# B&R Automation Studio project TD52 (part 31)

#### TrP_red.st
```iecst
(*******************************************************************************
TransP_red	Powerreduction cause of transformer warning

This code is confidential and proprietary to the INNIO Company.
It may not be used in any form, or reproduced in any manner,
without the express written permission of the INNIO Company.
Copyright, INNIO Company, 2019

Customized modifications: -
------------------------

History:
-------
V4.03.00	24.07.2015	Plattner Johannes
V4.04.00	23.09.2016	lettenb.	OUT_AG.rP_Red_TransformerWarning_Norm: /100 removed, bugfix
			08.05.2017				Pred logic corr., bugfix

Instructions for use:
--------------------

Power reduction from Transformer Warning.
Activates with parameter:		AuxiliariesGeneral::AsGlobalPV.bP_Red_TransformerWarning
Power setpoint with parameter:	AuxiliariesGeneral::AsGlobalPV.rP_Red_TransformerWarning_Rate

Outstandings:
------------
*******************************************************************************)
PROGRAM _CYCLIC

	(* Transformer power reduction aktive*)
	(*----------------------------------------------------------------------------*)
	IF Para.bP_Red_TransformerWarning_Sel AND NOT IN_AG.tTransformerWarning.Di THEN

		OUT_AG.rP_Red_TransformerWarning_Norm	:= LIMIT(0.5, Para.rP_Red_TransformerWarning_Rate,1.0);
		OUT_AG.bP_Red_TransformerWarning_Sel	:= TRUE;
	(*----------------------------------------------------------------------------*)

	(* Transformer power reduction inaktive*)
	(*----------------------------------------------------------------------------*)
	ELSE

		OUT_AG.bP_Red_TransformerWarning_Sel	:= FALSE;
		OUT_AG.rP_Red_TransformerWarning_Norm	:= 1.0;

	END_IF;
	(*----------------------------------------------------------------------------*)

END_PROGRAM
```

### Program Logical/AuxiliariesGeneral/Cnt_EO (IEC, version 4.13.0) - engine oil counter

#### Cnt_EOCyclic.st
```iecst
(***********************************************************************************************************************
AGGR: oil consumption counting and saving data (cyclic)

This code is confidential and proprietary to the INNIO Company.
It may not be used in any form, or reproduced in any manner, without the express
written permission of the INNIO Company.
Copyright, INNIO Company, 2024

- detection of oilcounter impulses
- logging oil volume(ml) and active energy(kwh)

Customized modifications: -
------------------------

History:
-------
V2.0	26.06.2007	TinelloM 	erstellt
V2.1	16.08.2007 	TinelloM 	überarbeitet
V2.3	31.03.2008 	TinelloM	überarbeitet für Serie
V3.20	20.07.2010	KoppM		anpassung für BR9 und analogen Füllstandsensor
V3.20.1	08.02.2011	TinelloM	IF ucIndexOil >1...
V3.90.0	06.12.2011	Ganguly		generated from oilcountCyclic.st V3.20.1
V3.90.1	12.03.2012	Denk		review and clean-up
V3.91	03.09.2013	Zengerer 	BUGFIX in nextline copy : OilCounter[i]	:= OilCounter[i+1];
V3.99.0 04.12.2013	lettenb.	slOilCounterMax,rSumOilVolume,rSumActiveEnergy: conversion dint_to_real added
V4.00.0	03.11.2014	lettenb.	init: DatObjCreate_01.MemType:= doSYSROM --> doUSRROM (vis kann bei update nicht in SYSROM schreiben)
		28.04.2015				set rAvgVolumeEnergy:=0 IF no averaging is selected, bugfix
V4.03.0	03.11.2015	lettenb.	calc. rAvgVolumeEnergy corr., bugfix
		11.01.2016				MM2VIS oil counter interfaces moved from Vis_AG -> Cnt_EO(to enable scroll function of settings)bugfix
		15.02.2016  waldhart	datenpunkte für HMI aus der IF-schleife entfernt(P19 test)
V4.05.0	14.12.2017	lettenb.	IN_AG.rP_Act_Norm_Filt -> IN_AG.rP_Act_Norm_Filt_TC2, mapping cleanup
		27.12.2017				bReset_Bh added, to reset oil counter memory after engine change(iCnt_OpHours -> 0)
V4.06.0 005 11.09.2018 Zengerer	beta: OUT_AG.tAG2PB.bPermSetupOk... new: transmit perm status info in InitUp
V4.07				Zengerer	Do not allow old data file lengt in init, to force rebuild with latest file format !
V4.09.0	09.10.2019	Schmid		BU1: reduced number of perm file write cycles (max every 10min)
V4.10.0	03.12.2020	Perktold,	added oil and coolant management
		25.01.2021	Schmid		bugfix oil refill blockade after iCnt_OpHours reset (engine exchange)
		11.03.2021	lettenb.	9004->9048, Msg# already used, bugfix
V4.11.0	19.01.2022	Schmid		option for oil sampling interval from oil quality sensor
V4.12.0	29.03.2023	Tinello		bugfix #1092 oil counter reset
V4.13.0	13.02.2024	Tinello		oil refill monitoring

Instructions for use:
--------------------
The parameter are stored in a data module which is stored on flash memory.
At start up the parameter will be readed from the flash memory and copied to

Outstandings:
------------
-
***********************************************************************************************************************)

PROGRAM _CYCLIC

(* getting time of the controller *)
	DTGetTime_RPS.enable := TRUE;							(* getting *)
	DTGetTime_RPS();
	DT_TO_DTStructure(DTGetTime_RPS.DT1, ADR(tRealTime));	(* change format *)
	DTGetTime_RPS.status;

	(* oil counter is active *)
	IF Para.b_OilActive THEN

		(* oilcounter impulse detection *)
		xR_TRIG_OilCounterImpulse(CLK := IN_AG.tCnt_OilPulse.Di);
		IF xR_TRIG_OilCounterImpulse.Q THEN  slOilCounterImpulse := slOilCounterImpulse + 1;	END_IF

		(* reset *)
		IF ucResetRegister1 = 0	THEN slOilCounterImpulse := 0;	END_IF

		(* oilcounter impulse detection for X20DC2395 --> Reset not possible *)
		IF REAL_TO_UINT(IN_AG.tCnt_Oil_DC2395.Ai) >= usOilCounterStart	THEN
			slOilCounterCircle	:= (REAL_TO_DINT(IN_AG.tCnt_Oil_DC2395.Ai) - usOilCounterStart) / 2;
		ELSE
			slOilCounterCircle	:= (REAL_TO_DINT(IN_AG.tCnt_Oil_DC2395.Ai) - usOilCounterStart + 65535) / 2;
		END_IF

		(* generate second based clock pulse *)
		xTON_SecondTick(IN := NOT xTON_SecondTick.Q, PT := T#980ms);		(* 980ms + 2 times cycle time = 1 sec.*)

		IF xTON_SecondTick.Q THEN

			(* reset *)
			bErrMsOilCounter	:= FALSE;
			b_OilRefillBlocked	:= FALSE;

			FOR i:=0 TO 19 BY 1 DO
				IF IN_AG.iCnt_OpHours > 0 AND IN_AG.iCnt_OpHours + 10000 < OilCounter[i].Bh THEN bReset_Bh := TRUE; (* reset OpHours(engine change)*)
				END_IF;
			END_FOR;

			(* Delete circular puffer array of oil measurements *)
			IF bReset_Bh THEN
				FOR i:=0 TO 19 BY 1 DO
					OilCounter[i].oil_volume		:= 0;
					OilCounter[i].delta_kwh 		:= 0;
					OilCounter[i].day 				:= 0;
					OilCounter[i].month 			:= 0;
					OilCounter[i].year 				:= 0;
					OilCounter[i].hour 				:= 0;
					OilCounter[i].minute 			:= 0;
					OilCounter[i].averaging			:= 0;
					OilCounter[i].Bh				:= 0;
					OilCounter[i].rOC_Consum		:= 0;
					OilCounter[i].rOC_DeltaOpHour	:= 0;
					OilCounter[i].rP_OC_Avg			:= 0;
				END_FOR

				ucIndexOil 	:= 0;										(* reset circular puffer index	*)
				bReset_Bh	:= FALSE;
			END_IF

			(* Identification of active oil counter input *)
			slOilCounterMax	:= MAX(slOilCounterCircle, slOilCounterImpulse);
			slOilCounterMax	:= REAL_TO_DINT(MAX(DINT_TO_REAL(slOilCounterMax), IN_AG.tCnt_Oil_NC150.Ai));

			slOilCounter	:= slOilCounterMax * 					(* maximum number of oil counter impulses 		*)
						   	   Para.iNum_OilPulse;					(* 1 impulse e.g.=2ml, -> 500 impulses/liter	*)

			(* Oil refill monitoring *)
			rVol_OilRefill_Max		:= (Para.rVol_OilRefill_Pct_EO_Level * 1000)	  *		(* oil refill volume [ml] per % oil level *)
									   (Para.r_OV_LimClose - Para.r_OV_LimOpen) * 100 *		(* % oil level between open- and closing of valve *)
									   (1.0 + Para.rPc_OilRefill_VolTolerance);				(* Tolerance *)

			bAMM_Vol_OilRefill_Hi	:= (slOilCounter > REAL_TO_DINT(rVol_OilRefill_Max)) AND Para.bOilRefill_MonAct AND Para.bEO_Level_Active;		(* W9378 *)

			(* calculation of kilowatt hour *)
			IF (IN_AG.rP_Act_Norm_Filt_TC2 * IN_AG.rP_Nom) > 50	THEN
				kwh	:= kwh + ((IN_AG.rP_Act_Norm_Filt_TC2 * IN_AG.rP_Nom) / 3600 );
			END_IF

			(* When Oilrefillvalve is closed, data will be saved *)
		 	xF_TRIG_OilRefillValve(CLK := OUT_AG.tEOVal_DemOpen.Do);

		 	IF 	xF_TRIG_OilRefillValve.Q	THEN
				(* monitoring measurement signal oil counter *)
				IF slOilCounter < 20 THEN	bErrMsOilCounter := TRUE;	END_IF

				(* Save oil data *)
				IF ucIndexOil >= 20 THEN
					(*----------------------------------------------------------------------------------*)
					(* After 20 measurements the data will be copied, so that the actual measurement	*)
					(* is allways shown in the last line.	 											*)
					(*----------------------------------------------------------------------------------*)
					FOR i:=0 TO 18 BY 1 DO
						OilCounter[i]			 		:= OilCounter[i+1];
//						OilCounter[i].oil_volume 		:= OilCounter[i+1].oil_volume;
//						OilCounter[i].delta_kwh			:= OilCounter[i+1].delta_kwh;
//						OilCounter[i].day				:= OilCounter[i+1].day;
//						OilCounter[i].month				:= OilCounter[i+1].month;
//						OilCounter[i].year				:= OilCounter[i+1].year;
//						OilCounter[i].hour				:= OilCounter[i+1].hour;
//						OilCounter[i].minute			:= OilCounter[i+1].minute;
//						OilCounter[i].averaging			:= OilCounter[i+1].averaging;
//						OilCounter[i].Bh				:= OilCounter[i+1].Bh;
					END_FOR

					OilCounter[19].oil_volume 			:= slOilCounter;		(* Save	actual measurement	*)
					OilCounter[19].delta_kwh			:= REAL_TO_DINT(kwh);
					OilCounter[19].day					:= USINT_TO_INT(tRealTime.day);
					OilCounter[19].month				:= USINT_TO_INT(tRealTime.month);
					OilCounter[19].year					:= UINT_TO_INT(tRealTime.year);
					OilCounter[19].hour 				:= USINT_TO_INT(tRealTime.hour);
					OilCounter[19].minute    			:= USINT_TO_INT(tRealTime.minute);
					OilCounter[19].averaging			:= TRUE;
					OilCounter[19].Bh					:= IN_AG.iCnt_OpHours;
				ELSE
					OilCounter[ucIndexOil].oil_volume 	:= slOilCounter;		(* Save	actual measurement	*)
					OilCounter[ucIndexOil].delta_kwh	:= REAL_TO_DINT(kwh);
					OilCounter[ucIndexOil].day			:= USINT_TO_INT(tRealTime.day);
					OilCounter[ucIndexOil].month		:= USINT_TO_INT(tRealTime.month);
					OilCounter[ucIndexOil].year			:= UINT_TO_INT(tRealTime.year);
					OilCounter[ucIndexOil].hour	 		:= USINT_TO_INT(tRealTime.hour);
					OilCounter[ucIndexOil].minute		:= USINT_TO_INT(tRealTime.minute);
					OilCounter[ucIndexOil].averaging	:= TRUE;
					OilCounter[ucIndexOil].Bh			:= IN_AG.iCnt_OpHours;

					ucIndexOil 	:= ucIndexOil + 1;								(* increase Index	*)
				END_IF

				(* reset kwh and oil counter	*)
				kwh 				:= 0;										(* reset kwh *)
				ucResetRegister1	:= 0;										(* Reset Counter(NC150)	*)
				usOilCounterStart 	:= REAL_TO_UINT(IN_AG.tCnt_Oil_DC2395.Ai);	(* initial Value *)

			ELSE
				ucResetRegister1	:= 128; 									(* binär 10000000 *)

				(* get oil counter settings from vis *)
				FOR i:=0 TO 19 BY 1 DO
					OilCounter[i].averaging	:= MM2VIS.tEO_Counter[i].averaging;
				END_FOR;

			END_IF

			(* oil counter values to vis *)
			FOR i:=0 TO 19 BY 1 DO
					MM2VIS.tEO_Counter[i].oil_volume		:= OilCounter[i].oil_volume;
					MM2VIS.tEO_Counter[i].delta_kwh 		:= OilCounter[i].delta_kwh;
					MM2VIS.tEO_Counter[i].day 				:= OilCounter[i].day;
					MM2VIS.tEO_Counter[i].month 			:= OilCounter[i].month;
					MM2VIS.tEO_Counter[i].year 				:= OilCounter[i].year;
					MM2VIS.tEO_Counter[i].hour 				:= OilCounter[i].hour;
					MM2VIS.tEO_Counter[i].minute 			:= OilCounter[i].minute;
					MM2VIS.tEO_Counter[i].Bh				:= OilCounter[i].Bh;
					MM2VIS.tEO_Counter[i].rOC_DeltaOpHour	:= OilCounter[i].rOC_DeltaOpHour;
					MM2VIS.tEO_Counter[i].rP_OC_Avg			:= OilCounter[i].rP_OC_Avg;
					MM2VIS.tEO_Counter[i].rOC_Consum		:= OilCounter[i].rOC_Consum;

					MM2VIS.tEO_Counter[i].averaging			:= OilCounter[i].averaging;
			END_FOR;

			(* averaging *)
			rSumOilVolume		:= 0;											(* reset sum of oil volume		*)
			rSumActiveEnergy	:= 0;											(* reset sum of active energy	*)
			rSumVolumeEnergy	:= 0;											(* reset sum of active volume/energy	*)
			ssAveragingNumber	:= 0;											(* reset averaging number		*)

			FOR i:=0 TO 19 BY 1	DO
				IF OilCounter[i].averaging	THEN
					rSumOilVolume		:= rSumOilVolume     + DINT_TO_REAL(OilCounter[i].oil_volume);	(* sum of oil volume	*)
					rSumActiveEnergy 	:= rSumActiveEnergy  + DINT_TO_REAL(OilCounter[i].delta_kwh);	(* sum of active energy	*)
					rSumVolumeEnergy 	:= rSumVolumeEnergy  + OilCounter[i].rOC_Consum;				(* sum of active consumption *)
					ssAveragingNumber	:= ssAveragingNumber + 1;										(* averaging number	*)
				END_IF
			END_FOR

			IF ssAveragingNumber = 0	THEN										(* DIVISION by zero *)
				rAvgOilVolume		:= 0;											(* No averaging	*)
				rAvgActiveEnergy  	:= 0;											(* No averaging	*)
				rAvgVolumeEnergy  	:= 0;											(* No averaging	*)
			ELSE
				rAvgOilVolume 		:= rSumOilVolume	/ ssAveragingNumber;		(* average over oil volume		*)
				rAvgActiveEnergy	:= rSumActiveEnergy / ssAveragingNumber;		(* average over active energy	*)
				IF rAvgActiveEnergy > 0.0 THEN
					rAvgVolumeEnergy	:= rAvgOilVolume * 0.89 / rAvgActiveEnergy; (* average over active oil volume / energy *)
				END_IF;
			END_IF;

			(* last measurement oil data for DIA.NE VIS trend and array for DIA.NE VIS picture OilCounter *)
			IF ucIndexOil = 0	THEN
				rVol_OC			:= DINT_TO_REAL(OilCounter[0].oil_volume);		(* oil volume during the last measurement 			*)
				rP_OC_Energy 	:= DINT_TO_REAL(OilCounter[0].delta_kwh);		(* active energy during the last measurement 		*)
				slOilRefill_Bh	:= OilCounter[0].Bh;							(* operating hour up to the time of last oil refill	*)
				rOC_DeltaOpHour:= 0;											(* operating hours during the last measurement		*)
				rP_OC_Avg		:= 0;											(* average power during the last measurement		*)

				IF 	OilCounter[0].delta_kwh = 0 THEN									(* DIVISION by zero *)
					rOC_Consum	:= 0;
				ELSE
					rOC_Consum	:= DINT_TO_REAL(OilCounter[0].oil_volume) * 0.89 / 		(* oil consumption during 	*)
								   DINT_TO_REAL(OilCounter[0].delta_kwh);				(* the last measurement		*)
				END_IF
				OilCounter[0].rOC_Consum := rOC_Consum;									(* operating hours during last measurement for VIS picture *)
			ELSE
				rVol_OC			:= DINT_TO_REAL(OilCounter[ucIndexOil-1].oil_volume);	(* oil volume during the last measurement 	*)
				rP_OC_Energy	:= DINT_TO_REAL(OilCounter[ucIndexOil-1].delta_kwh);	(* active energy during last measurement 	*)
				slOilRefill_Bh	:= OilCounter[ucIndexOil-1].Bh;							(* operating hour up to the last oil refill	*)
				IF ucIndexOil >1 THEN
					rOC_DeltaOpHour		:= DINT_TO_REAL(OilCounter[ucIndexOil-1].Bh -	(* operating hours during last measurement	*)
								       	   OilCounter[ucIndexOil-2].Bh);
					OilCounter[ucIndexOil-1].rOC_DeltaOpHour := rOC_DeltaOpHour;		(* operating hours during last measurement for VIS picture *)
				END_IF

				IF rOC_DeltaOpHour = 0 THEN									(* DIVISION by zero *)
					rP_OC_Avg	:= 0;
				ELSE
					rP_OC_Avg	:= rP_OC_Energy / rOC_DeltaOpHour;			(* Average power during last measurement *)
				END_IF
				OilCounter[ucIndexOil-1].rP_OC_Avg	:= rP_OC_Avg;			(* Average power during last measurement for VIS picture *)

				IF 	OilCounter[ucIndexOil-1].delta_kwh = 0 THEN				(* DIVISION by zero *)
					rOC_Consum	:= 0;
				ELSE
					rOC_Consum	:= DINT_TO_REAL(OilCounter[ucIndexOil-1].oil_volume) * 0.89 /
								   DINT_TO_REAL(OilCounter[ucIndexOil-1].delta_kwh);
				END_IF
				OilCounter[ucIndexOil-1].rOC_Consum	:= rOC_Consum;			(* operating hours during last measurement for VIS picture *)
			END_IF

			(* Blocking oil refill for X operating hours *)
			xCTU_OilRefillBlocked(CU:= (IN_AG.iCnt_OpHours = iOpH_OilRefillBlockPulse + 1), RESET:= xF_TRIG_OilRefillValve.Q, PV:= DINT_TO_UINT(Para.i_OilRefillBlocked));
			iOpH_OilRefillBlockPulse := IN_AG.iCnt_OpHours;
			IF IN_AG.iCnt_OpHours < (slOilRefill_Bh + Para.i_OilRefillBlocked) AND NOT xCTU_OilRefillBlocked.Q AND IN_AG.tEO_Level_Lo_TC2.Di AND NOT bEO_Level_Lo THEN
				b_OilRefillBlocked	:= TRUE;
			END_IF

			(* calculated oil counter values to vis *)
			MM2VIS.rVol_OC_Avg			:= rAvgOilVolume;
			MM2VIS.rOC_Energy_Avg		:= rAvgActiveEnergy;
			MM2VIS.rP_OC_Energy			:= rP_OC_Energy;
			MM2VIS.rP_OC_Avg			:= rP_OC_Avg;
			MM2VIS.rOC_DeltaOpHour		:= rOC_DeltaOpHour;
			MM2VIS.rOC_Consum			:= rOC_Consum;
			MM2VIS.rVol_OC				:= rVol_OC;
			MM2VIS.rOC_Consum_Avg		:= rAvgVolumeEnergy;

		END_IF

		(*----------------------------------------------------------------------------------------*)
		(* save oil counter values in permanent memory *)

		(* 10 seconds timer *)
		xTON_WritePMEM(IN := NOT xTON_WritePMEM.Q, PT:= T#10s);
		xTON_BlockMinFileAge(IN := bBlock_MinFileAge, PT:= T#10m);
		IF xTON_BlockMinFileAge.Q THEN	bBlock_MinFileAge := FALSE; END_IF;

		(* every 10 seconds or at write once the parameter values are copied to the structure pm *)
		IF xTON_WritePMEM.Q OR write_once THEN

			(* ------------- V1.10 ---------------- *)
			pmOil.kwh				:= kwh;				(* copy parameter value to structure pm *)
			pmOil.ucIndexOil		:= ucIndexOil;		(* ----------------- " ---------------- *)
			pmOil.OilCounter		:= OilCounter;

		END_IF;

		(* cyclic calcualtion of parameter checksum	*)
		IF xTON_WritePMEM.Q THEN
			ulChecksum := 0;

			FOR ulPMPointer := ADR(pmOil) TO (ADR(pmOil) + pm_len - SIZEOF(ulChkValue)) DO
				memcpy(ADR(ulChkValue), ulPMPointer, SIZEOF(ulChkValue));
				ulChecksum := (ulChecksum XOR ulChkValue)+ulChkValue;
			END_FOR;

			IF ulChecksumOld <> ulChecksum THEN					(* if checksum has changed 		*)
				ulChecksumOld := ulChecksum;					(* save last cheksum value		*)
				bWriteDataObj := TRUE;							(* set flag for write checksum	*)
			END_IF;

		END_IF

		(* write structure pm to the permanent memory module *)
		IF ( (bWriteDataObj AND NOT bBlock_MinFileAge) OR write_once ) THEN

			DatObjWrite_01();									(* run data object write fub 					*)

			IF DatObjWrite_01.status <> ERR_FUB_BUSY THEN		(* wait if data object write fub is busy 		*)
				bWriteDataObj 	:= FALSE;						(* reset data object write flag					*)
				write_once 		:= FALSE;						(* reset write_once flag 						*)
				iPM_WriteCnt 	:= iPM_WriteCnt + 1;			(* counter for done data object module writes	*)

				IF OUT_AG.tAG2PB.iPermStatus >=0 THEN 												(* new V4.06: if not already on error state, then transmit this perm status info *)
					OUT_AG.tAG2PB.iPermStatus := LIMIT(2, OUT_AG.tAG2PB.iPermStatus + 1, 999);		(* new V4.06: transmit OK= positive perm status info *)
					IF OUT_AG.tAG2PB.iPermStatus = 999 THEN OUT_AG.tAG2PB.iPermStatus := 2; END_IF;	(* new V4.06: transmit OK= positive perm status info *)
					OUT_AG.tAG2PB.bPermSetupOk := TRUE;												(* new V4.06: transmit perm status info *)
				END_IF;

				IF DatObjWrite_01.status = ERR_NOERROR THEN		(* if status = NO ERROR -> block further write requests for 10min to avoid CF wear down	*)
					bBlock_MinFileAge := TRUE;
				ELSE											(* if error status not no error 				*)
					pm_Error := 1005;  //:= 4;					(* set data object write error state			*)
				END_IF;
			END_IF;

		END_IF;

	ELSE
		(* Reset *)
		bErrMsOilCounter		:= FALSE;
		b_OilRefillBlocked		:= FALSE;
		bAMM_Vol_OilRefill_Hi	:= FALSE;
	END_IF;

	(* set RPS warning if no access to SysRom file is possible *)
	TON_WarnDelay(IN := pm_Error > 0 , PT:= T#15s);
	IF TON_WarnDelay.Q AND (OUT_AG.tAG2PB.iPermStatus >= 0) THEN 	OUT_AG.tAG2PB.iPermStatus := LIMIT(-999999,-UINT_TO_DINT(pm_Error) ,-1)	;	END_IF	(* new V4.06: transmit error as negative perm status info *)
	IF (OUT_AG.tAG2PB.iPermStatus < 0) THEN 	OUT_AG.tAG2PB.bPermSetupOk := FALSE	;	END_IF		(* No reset of error bit - every error needs reboot *)		(* new V4.06: transmit perm status info *)

(*Start Oil & Coolant Management*)
	IF IN_AG.tPB2MM.bParaSetupOk AND (Para.bEO_Management_Active OR Para.bCW_Management_Active) THEN
		xTP_OilExchange.IN			:= FALSE;													(*Reset TP FUB Input*)
		xTP_OilSample.IN			:= FALSE;													(*Reset TP FUB Input*)
		xTP_CWExchange.IN			:= FALSE;													(*Reset TP FUB Input*)
		xTP_CWSample.IN				:= FALSE;													(*Reset TP FUB Input*)

(*Oil-Part*)
		IF Para.bEO_Management_Active THEN														(*if the oil management function is active then*)

			IF (IN_AG.iCnt_OpHours = (iCnt_OpHours_old + 1)) THEN								(*if engine Oh increase by 1 then*)
				MM2VIS.iCnt_OilOh 			:= MM2VIS.iCnt_OilOh + 1;							(*increase oil operating hour counter by one*)
				MM2VIS.iCnt_OilSampleOh		:= MM2VIS.iCnt_OilSampleOh - 1;						(*decrease oil sample counter by one*)
			END_IF;

			IF VIS2MM.bOilExchange THEN															(*if Button "Oil exchanged" pressed on HMI then*)
				MM2VIS.tLastOilExchange.Oh_fluid	:= MM2VIS.iCnt_OilOh;						(*Save oil operation hours at exchange*)
				MM2VIS.tLastOilExchange.Oh_engine	:= IN_AG.iCnt_OpHours;						(*Save engine operation hours at exchange*)
				MM2VIS.tLastOilExchange.day			:= USINT_TO_INT(tRealTime.day);				(*Save date at exchange*)
				MM2VIS.tLastOilExchange.month		:= USINT_TO_INT(tRealTime.month);			(*Save date at exchange*)
				MM2VIS.tLastOilExchange.year		:= UINT_TO_INT(tRealTime.year);				(*Save date at exchange*)
				MM2VIS.iCnt_OilOh					:= 0;										(*Reset oil counter to zero*)
				IF VIS2MM.bOQS_OilSampleOh_Man THEN
					MM2VIS.iCnt_OilSampleOh			:= VIS2MM.iOilSampleOh;						(*Reset oil sample counter - Manual interval*)
				ELSE
					MM2VIS.iCnt_OilSampleOh			:= MM2VIS.iOQS_OilSampleOh;					(*Reset oil sample counter - Automatic interval from oil quality sensor*)
				END_IF;
				xTP_OilExchange.IN					:= TRUE;									(*Trigger operation message "Oil exchanged"*)
				VIS2MM.bOilExchange 				:= FALSE;									(*Reset Button "Oil exchanged" on HMI*)
			END_IF;

			xTP_OilExchange();																	(*Execute FUB for operatin message*)

			IF VIS2MM.bOilSample THEN
				IF VIS2MM.bOQS_OilSampleOh_Man THEN
					MM2VIS.iCnt_OilSampleOh			:= VIS2MM.iOilSampleOh;						(*Reset oil sample counter - Manual interval*)
				ELSE
					MM2VIS.iCnt_OilSampleOh			:= MM2VIS.iOQS_OilSampleOh;					(*Reset oil sample counter - Automatic interval from oil quality sensor*)
				END_IF;
				MM2VIS.tLastOilSample.Oh_fluid		:= MM2VIS.iCnt_OilOh;						(*Save oil operation hours when sample was taken*)
				MM2VIS.tLastOilSample.Oh_engine		:= IN_AG.iCnt_OpHours;						(*Save engine operation hours when sample was taken*)
				MM2VIS.tLastOilSample.day			:= USINT_TO_INT(tRealTime.day);				(*Save date when sample was taken*)
				MM2VIS.tLastOilSample.month			:= USINT_TO_INT(tRealTime.month);			(*Save date when sample was taken*)
				MM2VIS.tLastOilSample.year			:= UINT_TO_INT(tRealTime.year);				(*Save date when sample was taken*)
				xTP_OilSample.IN					:= TRUE;									(*Trigger operation message "Oil sample taken"*)
				VIS2MM.bOilSample 					:= FALSE;									(*Reset Button "Oil sample taken" on HMI"*)
			END_IF;

			xTP_OilSample();																	(*Execute FUB for operating message*)

			bMsg9332_set		:= (MM2VIS.iCnt_OilSampleOh < 1) AND (IN_AG.iCnt_OpHours > 0);	(*set warning to take oil sample*)

			IF VIS2MM.iOilSampleOh = 0 THEN VIS2MM.iOilSampleOh := 150; END_IF;					(*initialize oil sample intervall in case value is zero*)

		ELSE																					(*if the oil management function is NOT active then*)

			xTP_OilExchange();																	(*Execute FUB for operatin message*)
			xTP_OilSample();																	(*Execute FUB for operating message*)
			bMsg9332_set			:= FALSE;													(*Reset warning "take oil sample"*)
			VIS2MM.bOilExchange 	:= FALSE;													(*Reset HMI button "oil exchanged"*)
			VIS2MM.bOilSample 		:= FALSE;													(*Reset HMI button "oil sample taken"*)
		END_IF;
(*Coolant-Part*)
		IF Para.bCW_Management_Active THEN														(*if the coolant management function is active then*)

			IF (IN_AG.iCnt_OpHours = (iCnt_OpHours_old + 1)) THEN								(*if engine Oh increase by 1 then*)
				MM2VIS.iCnt_CWOh 			:= MM2VIS.iCnt_CWOh + 1;							(*increase cooling water operating hour counter by one*)
				MM2VIS.iCnt_CWSampleOh		:= MM2VIS.iCnt_CWSampleOh - 1;						(*decrease cooling water sample counter by one*)
			END_IF;

			IF VIS2MM.bCWExchange THEN															(*Button "Cooling water exchanged" pressed on HMI *)
				MM2VIS.tLastCWExchange.Oh_fluid		:= MM2VIS.iCnt_CWOh;						(*Save cooling water operation hours at exchange*)
				MM2VIS.tLastCWExchange.Oh_engine	:= IN_AG.iCnt_OpHours;						(*Save engine operation hours at exchange*)
				MM2VIS.tLastCWExchange.day			:= USINT_TO_INT(tRealTime.day);				(*Save date at exchange*)
				MM2VIS.tLastCWExchange.month		:= USINT_TO_INT(tRealTime.month);			(*Save date at exchange*)
				MM2VIS.tLastCWExchange.year			:= UINT_TO_INT(tRealTime.year);				(*Save date at exchange*)
				MM2VIS.iCnt_CWOh					:= 0;										(*Reset cooling water counter to zero*)
				MM2VIS.iCnt_CWSampleOh				:= VIS2MM.iCWSampleOh;						(*Reset cooling water sample counter*)
				xTP_CWExchange.IN					:= TRUE;									(*Trigger operation message "Cooling water exchanged"*)
				VIS2MM.bCWExchange 					:= FALSE;									(*Reset Button "Cooling water exchanged" on HMI*)
			END_IF;

			xTP_CWExchange();																	(*Execute FUB for operatin message*)

			IF VIS2MM.bCWSample THEN
				MM2VIS.iCnt_CWSampleOh				:= VIS2MM.iCWSampleOh;						(*Reset cooling water sample counter*)
				MM2VIS.tLastCWSample.Oh_fluid		:= MM2VIS.iCnt_CWOh;						(*Save cooling water operation hours when sample was taken*)
				MM2VIS.tLastCWSample.Oh_engine		:= IN_AG.iCnt_OpHours;						(*Save engine operation hours when sample was taken*)
				MM2VIS.tLastCWSample.day			:= USINT_TO_INT(tRealTime.day);				(*Save date when sample was taken*)
				MM2VIS.tLastCWSample.month			:= USINT_TO_INT(tRealTime.month);			(*Save date when sample was taken*)
				MM2VIS.tLastCWSample.year			:= UINT_TO_INT(tRealTime.year);				(*Save date when sample was taken*)
				xTP_CWSample.IN						:= TRUE;									(*Trigger operation message "Cooling water sample taken"*)
				VIS2MM.bCWSample 					:= FALSE;									(*Reset Button "Cooling water sample taken" on HMI"*)
			END_IF;

			xTP_CWSample();																		(*Execute FUB for operating message*)

			bMsg9333_set		:= (MM2VIS.iCnt_CWSampleOh < 1) AND (IN_AG.iCnt_OpHours > 0);	(*set warning to take cooling water sample*)

			IF VIS2MM.iCWSampleOh = 0 THEN VIS2MM.iCWSampleOh := 2000; END_IF;					(*initialize cooling water sample intervall in case value is zero*)

		ELSE																					(*if the coolant management function is NOT active then*)

			xTP_CWExchange();																	(*Execute FUB for operatin message*)
			xTP_CWSample();																		(*Execute FUB for operating message*)
			bMsg9333_set			:= FALSE;													(*Reset warning "take coolant sample"*)
			VIS2MM.bCWExchange	 	:= FALSE;													(*Reset HMI button "coolant exchanged"*)
			VIS2MM.bCWSample 		:= FALSE;													(*Reset HMI button "coolant sample taken"*)
		END_IF;
(*Oil & Coolant*)
		iCnt_OpHours_old		:= IN_AG.iCnt_OpHours;											(*save engine Oh for next cycle*)

	ELSE																						(*if both functions (oil & coolant management) are NOT active*)

		iCnt_OpHours_old		:= IN_AG.iCnt_OpHours;											(*save engine Oh for next cycle*)
		bMsg9332_set			:= FALSE;														(*Reset warning "take oil sample"*)
		VIS2MM.bOilExchange 	:= FALSE;														(*Reset HMI button "oil exchanged"*)
		VIS2MM.bOilSample 		:= FALSE;														(*Reset HMI button "oil sample taken"*)

		bMsg9333_set			:= FALSE;														(*Reset warning "take coolant sample"*)
		VIS2MM.bCWExchange	 	:= FALSE;														(*Reset HMI button "coolant exchanged"*)
		VIS2MM.bCWSample 		:= FALSE;														(*Reset HMI button "coolant sample taken"*)

		xTP_OilExchange(IN:= FALSE);															(*Reset TP FUB Input*)
		xTP_OilSample(IN:= FALSE);																(*Reset TP FUB Input*)
		xTP_CWExchange(IN:= FALSE);																(*Reset TP FUB Input*)
		xTP_CWSample(IN:= FALSE);																(*Reset TP FUB Input*)

	END_IF;

	xTON_OilExchange.IN			:= xTP_OilExchange.Q;											(*delay 1.11s to ensure that the correct additional infos get stored with the operating message*)
	xTON_OilExchange();
	xTON_OilSample.IN			:= xTP_OilSample.Q;
	xTON_OilSample();

	bMsg9002_set				:= xTON_OilExchange.Q;											(*set B9002 Oil exchanged*)
	bMsg9001_set				:= xTON_OilSample.Q;											(*set B9001 Oil sample taken*)

	xTON_CWExchange.IN			:= xTP_CWExchange.Q;											(*delay 1.11s to ensure that the correct additional infos get stored with the operating message*)
	xTON_CWExchange();
	xTON_CWSample.IN			:= xTP_CWSample.Q;
	xTON_CWSample();

	bMsg9048_set				:= xTON_CWExchange.Q;											(*set B9048 Coolant exchanged*)
	bMsg9003_set				:= xTON_CWSample.Q;												(*set B9003 Coolant sample taken*)

(*End Oil & Coolant Management*)

END_PROGRAM
```

#### Cnt_EOInit.st
```iecst
(*******************************************************************************
AGGR: oil consumption counting and saving data (init)

This code is confidential and proprietary to the INNIO Company.
It may not be used in any form, or reproduced in any manner, without the express
written permission of the INNIO Company.
Copyright, INNIO Company, 2019

- set some init parameters
- check for existing permanent memory data module
- if permanent memory data module doesn´t exists, or length of data module and
  parameter struct is different create permanent memory data module
- prepare parameter for permanent memory data write in cyclic task
- if permanent memory data module exist read data and copy to structure pm
- if permanent memory data module exist copy data from structure pm to program parameter

Customized modifications: -
------------------------

History:
-------
V2.30	31-03-2008	TinelloM,	generated from perm_par
V3.99.0	??						Add Metamodule name to_perm name
V3.99.1	06.11.2014	Zengerer	USERROM, changed from SYSROM due to VIS reasons
V4.06.0 005 05.10.2018 Zengerer beta: OUT_AG.tAG2PB.bPermSetupOk,  transmit perm status info, pm_Error +1000

Instructions for use:
--------------------
The parameter are stored in a data module which is stored on flash memory.
At start up the parameter will be readed from the flash memory and copied to
the parameter variables. If the data module does not exist or the length of
data module and parameter struct is different, the data module will be created.

Outstandings:
------------
*******************************************************************************)

PROGRAM _INIT

	(* set oil counter counting direction to positive *)
	ucModeRegister1 := 14;

	(* set some init parameters *)
	xTON_WritePMEM(IN := FALSE, PT:= T#10s);					(* reset used timer function blocks 			*)
	xTP_OilExchange.PT 	:= T#5s;
	xTP_OilSample.PT 	:= T#5s;
	xTP_CWExchange.PT 	:= T#5s;
	xTP_CWSample.PT 	:= T#5s;
	xTON_OilExchange.PT := T#1s500ms;
	xTON_OilSample.PT 	:= T#1s500ms;
	xTON_CWExchange.PT 	:= T#1s500ms;
	xTON_CWSample.PT 	:= T#1s500ms;

	pm_Error 	:= ERR_NOERROR;								(* reset permanent memory error	status			*)
	write_once 	:= FALSE;				 					(* reset flag for write permanent memory once	*)
	pm_len 		:= SIZEOF(pmOil);							(* define data length of permenent memory		*)
	strcpy(ADR(ModulName),ADR('AuxiliariesGeneral::oil_perm'));		(* define name of permanent memory data module	*)

	(* check for existing permanent memory data module	*)
	DatObjInfo_01.enable:= TRUE;							(* enable FUB									*)
	DatObjInfo_01.pName := ADR(ModulName);					(* set permanent memory data module name 		*)
	DatObjInfo_01();										(* run data object info FUB						*)

	(* check error status of data object info FUB	*)
	IF DatObjInfo_01.status = ERR_NOERROR THEN				(* if no error	--> permanent memory data module exists	*)
		pm_id 	:= DatObjInfo_01.ident;						(* copy permanent memory data module ident			*)
		pm_p 	:= DatObjInfo_01.pDatObjMem;				(* copy permanent memory data module memory adres	*)
	ELSE
		bCreateDataObj := TRUE;								(* set flag for create new data object	*)
		pm_Error := 1001;									(* set permanent memory error status	*)
	END_IF;

	(* check length of parameter struct with length of data object *)

	CASE DatObjInfo_01.len OF

//(*488:   perm_oil_vers  := 230;							(  488 = length of perm_par V2.30 !DISABELED! Do not allow old data files to force rebuild with latest file format !*)
//(*	   OUT_AG.tAG2PB.iPermStatus := OUT_AG.tAG2PB.iPermStatus + perm_oil_vers	;	( new V4.06: transmit perm status info *)
		// OUT_AG.tAG2PB.bPermSetupOk := TRUE	;				(* new V4.06: transmit perm status info *)

	728:   perm_oil_vers  := 390;							(* 728 = length of perm_par V3.90 *)
		   OUT_AG.tAG2PB.iPermStatus := OUT_AG.tAG2PB.iPermStatus + perm_oil_vers	;	(* new V4.06: transmit perm status info *)
		// OUT_AG.tAG2PB.bPermSetupOk := TRUE	;				(* new V4.06: transmit perm status info *)

	(* insert new perm_par Version here
	(* 		   bCreateDataObj := TRUE;						(* set flag for create new data object	*)
	(* xxxx:   perm_oil_vers  := yyy;						(* xxxx = length of perm_par Vy.yy *)

	ELSE
		bCreateDataObj := TRUE;								(* set flag for create new data object	*)
		OUT_AG.tAG2PB.bPermSetupOk := FALSE	;				(* new V4.06: transmit perm status info *)
		OUT_AG.tAG2PB.iPermStatus := OUT_AG.tAG2PB.iPermStatus  - 1000 ;			(*Perm Error*)
	END_CASE;

	(* if permanent memory data module exist read data and copy to structure pm	*)
	IF pm_Error = ERR_NOERROR THEN							(* permanent memory data module exist 				*)
		DatObjRead_01.enable 		:= TRUE;				(* enable read permanent memory module data 		*)
		DatObjRead_01.ident 		:= pm_id;				(* set identifier of permanent memory data module	*)
		DatObjRead_01.Offset 		:= 0;					(* start at memory offest zero 						*)
		DatObjRead_01.pDestination 	:= ADR(pmOil);			(* set permanent data destination adress			*)
		DatObjRead_01.len 			:= DatObjInfo_01.len;	(* set length of permanent data module				*)

		REPEAT	(* repeat until data of permanent memory data module have been read *)
			DatObjRead_01();								(* FUB read data from permanent data module 		*)
			UNTIL	DatObjRead_01.status <> ERR_FUB_BUSY	(* wait if FUB is busy 	*)
		END_REPEAT;

		IF DatObjRead_01.status <> ERR_NOERROR THEN			(* if status of read permanent data moduel is not OK 	*)
			pm_Error :=	1002;								(* set permanent memory error status					*)
		END_IF
	END_IF;

	(* if permanent memory data module exist --> copy data from structure pm to program parameter *)
	IF pm_Error = ERR_NOERROR THEN

		(* ------------- V2.30 ---------------- *)
		kwh						:= pmOil.kwh;
		ucIndexOil				:= pmOil.ucIndexOil;
		OilCounter				:= pmOil.OilCounter;

		(* ------------- V1.xx--------------- *)
		(* perm_oil_vers >= 240 THEN
		*)

		   IF OUT_AG.tAG2PB.iPermStatus >=0 THEN 													(* new V4.06: transmit perm status info *)
				OUT_AG.tAG2PB.iPermStatus := LIMIT(2, OUT_AG.tAG2PB.iPermStatus + pm_len, 999999);		(* new V4.06: transmit perm status info *)
		   		OUT_AG.tAG2PB.bPermSetupOk := TRUE	;												(* new V4.06: transmit perm status info *)
			END_IF																					(* new V4.06: transmit perm status info *)
	END_IF;

	(* create new permanent memory data module	*)
	IF bCreateDataObj THEN

		(* try to delete old data module *)
		DatObjDelete_PermMem.enable := TRUE;
		DatObjDelete_PermMem.ident 	:= pm_id;

		REPEAT	(* repeat until delete of permanent memory data module is ready *)
			DatObjDelete_PermMem();						(* FUB for delete permanent memory data module *)
			UNTIL	DatObjDelete_PermMem.status <> ERR_FUB_BUSY		(* wait if FUB is busy 	*)
		END_REPEAT;

		(* create new one *)
		DatObjCreate_01.enable	 := TRUE;				(* enable create permanent memory data module FUB 	*)
		DatObjCreate_01.grp 	 := 0;					(* must to be set to zero							*)
		DatObjCreate_01.pName 	 := ADR(ModulName);		(* set permanent memory data module name 			*)
		DatObjCreate_01.len 	 := pm_len;				(* set length ofpermanent memory data module		*)
		DatObjCreate_01.MemType  := doUSRROM;			(* create permanent memory data module at USERROM (changed from doSYSROM due to VIS reasons)	*)
		DatObjCreate_01.Option 	 := 0;					(* cyclic checksum monitoring is on					*)
		DatObjCreate_01.pCpyData := 0;					(* no data will be copied do the perm. mem. data module *)

		pm_Error:= 1003;								(* set permanent memory error status	*)

		REPEAT	(* repeat until generation of permanent memory data module is ready *)
			DatObjCreate_01();							(* FUB for create permanent memory data module 		*)
			UNTIL	DatObjCreate_01.status <> ERR_FUB_BUSY		(* wait if FUB is busy 	*)
		END_REPEAT;

		IF DatObjCreate_01.status = ERR_NOERROR THEN	(* is creation of permanent memory data module OK 	*)
			pm_p 	:= DatObjCreate_01.pDatObjMem;		(* set memory adress of permanent memory data module*)
			pm_id 	:= DatObjCreate_01.ident;			(* set identifier of permanent memory data module 	*)
		ELSE
			pm_Error:= 1004;							(* set permanent memory error status	*)
		END_IF;
	END_IF;

	(* prepare parameter for permanent memory data write in cyclic task *)
	IF pm_Error < 1004 THEN								(* permanent memory data module exist or has been created	*)
		DatObjWrite_01.enable 	:= TRUE;				(* enable permanent memory data module read FUB 	*)
		DatObjWrite_01.ident 	:= pm_id;				(* set identifier of permanent memory data module 	*)
		DatObjWrite_01.Offset 	:= 0;					(* start at memory offest zero 						*)
		DatObjWrite_01.pSource 	:= ADR(pmOil);			(* set permanent memory data module name 			*)
		DatObjWrite_01.len 		:= pm_len;				(* set length ofpermanent memory data module		*)
	END_IF;

	(* calcualte actual checksum of parameter structure	*)
	ulChecksumOld := 0;									(* reset checksum value *)

	FOR ulPMPointer := ADR(pmOil) TO (ADR(pmOil) + pm_len - SIZEOF(ulChkValue)) DO
		memcpy(ADR(ulChkValue), ulPMPointer, SIZEOF(ulChkValue));
		ulChecksumOld := ulChecksumOld XOR ulChkValue;
	END_FOR

	(**Forward Perm Error - new V4.06 *)
	IF (pm_Error > 0) AND (OUT_AG.tAG2PB.iPermStatus >= 0) THEN 	OUT_AG.tAG2PB.iPermStatus := LIMIT(-999999,-UINT_TO_DINT(pm_Error) ,-1)	;	END_IF		(* new V4.06: transmit error as negative perm status info *)
	IF (OUT_AG.tAG2PB.iPermStatus < 0) THEN 	OUT_AG.tAG2PB.bPermSetupOk := FALSE	;	END_IF			(* new V4.06: transmit perm status info *)

END_PROGRAM
```

#### Cnt_EO.var
```iecst
VAR
	write_once : BOOL; (*write permanent memory once *)
	bCreateDataObj : BOOL; (*TRUE=create new data object *)
	bWriteDataObj : BOOL; (*TRUE=write data object module *)
	DatObjCreate_01 : DatObjCreate; (*data object create *)
	DatObjDelete_PermMem : DatObjDelete; (*data object delete *)
	DatObjInfo_01 : DatObjInfo; (*data object info *)
	DatObjRead_01 : DatObjRead; (*data object read *)
	DatObjWrite_01 : DatObjWrite; (*data object write *)
	slOilCounterMax : DINT := 0; (*maximum number of oil counter impulses*)
	slOilCounter : DINT := 0; (*number of impulses from oil counter*)
	slOilCounterCircle : DINT := 0; (*number of impulses from oil counter --> calculated value*)
	xF_TRIG_OilRefillValve : F_TRIG := (0); (*FuB *)
	ssAveragingNumber : INT := 0; (*number of averaging*)
	i : INT := 0;
	pmOil : ParaOil_typ; (*permanent memory tags *)
	xR_TRIG_OilCounterImpulse : R_TRIG := (0); (*FuB*)
	rSumActiveEnergy : REAL := 0.0; (*sum of active energy*)
	rSumVolumeEnergy : REAL := 0.0; (*sum of active volume/energy*)
	rSumOilVolume : REAL := 0.0; (*sum of oil volume *)
	ModulName : STRING[35]; (*module name of object *)
	xTON_SecondTick : TON := (0); (*FuB*)
	xTON_WritePMEM : TON := (0); (*delay write permanent memory *)
	pm_len : UDINT; (*permanent value lenght *)
	pm_p : UDINT; (*permanent value pointer *)
	pm_id : UDINT; (*permanent value identifier *)
	ulChecksumOld : UDINT; (*last vlaue of parameter checksum *)
	ulChecksum : UDINT; (*parameter checksum value *)
	ulPMPointer : UDINT; (*adress of actual checksum value *)
	ulChkValue : UDINT; (*actual value of parameter pointer *)
	pm_Error : UINT; (*permanent value error *)
	perm_oil_vers : UINT; (*version*)
	usOilCounterStart : UINT := 0; (*oil counter initial value = value before refill*)
	DTGetTime_RPS : DTGetTime;
	ERR_NOERROR : UINT; (* status for no error *)
	bReset_Bh : BOOL;
	TON_WarnDelay : TON; (*V4.06*)
	xTON_BlockMinFileAge : TON;
	bBlock_MinFileAge : BOOL;
	iPM_WriteCnt : UINT; (*data module write counter *) (*old VarName: pmPrstWriteCnt*)
	xTP_OilExchange : TP;
	xTP_OilSample : TP;
	xTP_CWExchange : TP;
	xTP_CWSample : TP;
	xTON_OilExchange : TON;
	xTON_OilSample : TON;
	xTON_CWExchange : TON;
	xTON_CWSample : TON;
	iCnt_OpHours_old : DINT;
	xCTU_OilRefillBlocked : CTU;
	iOpH_OilRefillBlockPulse : DINT;
	rVol_OilRefill_Max : REAL := 0.0; (*Calculated oil refill volume maximum [ml]*)
END_VAR
```

### Program Logical/AuxiliariesGeneral/OilQsens (IEC, version 4.12.0) - Oil condition monitoring

#### OilQsensCyclic.st
```iecst
(*******************************************************************************
OilQsens	Oil condition monitoring (cyclic)

This code is confidential and proprietary to the INNIO Company.
It may not be used in any form, or reproduced in any manner, without the express
written permission of the INNIO Company.
Copyright, INNIO Company, 2019

- handle analog signals
- counter handling

Customized modifications: -
------------------------

History:
-------
V3.90.0	20.08.2013	Denk 		Created initial structured text code from V0.01.1
V4.11.0	05.11.2021	Schmid		new oil quality sensor with CAN readout added
V4.11.1	04.02.2022	Schmid		reworked CAN oil configuration for 2nd generation OQS
V4.11.2	22.02.2022	Schmid		oil quality sensor modifications from validation
V4.12.0	12.10.2022	Bacci		oil quality sensor modification in accordance with TANDELTA firmware 4.03. Para.rT_OQS_LimLo and MM2VIS.iOQS_OC_Status_Num added. General user experience improvement
V4.13.0 27.09.2023 	Bacci		Flucon sensor clean-up

Instructions for use:
--------------------
-

Outstandings:
------------
- Counter handling

*******************************************************************************)
PROGRAM _CYCLIC

(*TanDelta oil quality sensor*)
IF Para.iOQS_Config = 1 THEN

	IF VIS2MM.bOQS_OC_ConfigOilType THEN
		VIS2MM.bOQS_OC_ConfigOilType	:=	FALSE;
		iOQS_OC_ComState				:=	_CONFIG_OIL;
	END_IF;

	IF VIS2MM.bOQS_OC_ReadOilType THEN
		VIS2MM.bOQS_OC_ReadOilType		:=	FALSE;
		iOQS_OC_ComState				:=	_READ_CONFIG;
	END_IF;

	IF		VIS2MM.iOQS_OC_OilTypeIdx = 1 THEN		tOilConfig.sData_OilCfgUpd	:=	sStdOilCfg[1];
	ELSIF	VIS2MM.iOQS_OC_OilTypeIdx = 2 THEN		tOilConfig.sData_OilCfgUpd	:=	sStdOilCfg[2];
	END_IF;

	(*============================== CAN WRITE COMMANDS ===============================*)
	xCANwrite_OQS_OC.us_ident	:= IN_AG.iCAN_OQS_OC_us_ident;
	xCANwrite_OQS_OC.can_id		:= iSendMsgID_OC;
	xCANwrite_OQS_OC.data_adr	:= ADR(tDataSend_OC);
	xCANwrite_OQS_OC.data_lng	:= UDINT_TO_USINT(iDataLength_OC);

	IF iOQS_OC_ComState <> iOQS_OC_ComStateOld THEN
		bSend_OC			:= FALSE;
		iSendMsgCnt			:= 0;
	ELSE
		CASE iOQS_OC_ComState OF
			_READ_DATA:
				(*---------------------------- PREPARATION DATA REQUEST ----------------------------*)
				(* send data request *)
				IF iSendMsgCnt = 0 THEN
					iSendMsgCnt		:= 1;
					bSend_OC		:= TRUE;
				END_IF;
				IF bAck_OC THEN
					bSend_OC		:= TRUE;
					bAck_OC			:= FALSE;
				ELSIF xTON_AckMissing.Q THEN
					bSend_OC		:= TRUE;	// repeat send request
				END_IF;

				IF iSendMsgCnt < 4 THEN
					tDataSend_OC	:= tDataReq_OC;	// read data msg
					tDataSend_OC[3]	:= UINT_TO_BYTE(iSendMsgCnt);
				ELSE
					tDataSend_OC	:= tErrReq_OC;	// read error status msg
				END_IF;
				(*---------------------------- PREPARATION DATA REQUEST ----------------------------*)

			_CONFIG_OIL:
				(*---------------------------- BEGIN CONFIG OIL ---------------------------*)
				(* oil type reconfiguration *)
				(* write oil type configuration *)
				IF iSendMsgCnt = 0 THEN
					tDataSend_OC		:= tOilCfgWrite_Send_OC;
					tDataSend_OC[0]		:= tOilCfgWrite_SendB0_OC[iSendMsgCnt];

					xHexStr2ByteArr.iOffsetStrRd	:= 0;
					bSend_OC						:= TRUE;
				ELSE
					IF bAck_OC THEN
						bSend_OC	:= TRUE;
						bAck_OC		:= FALSE;

						xHexStr2ByteArr.pByteArray	:= ADR(tDataSend_OC[1]);
						xHexStr2ByteArr.pHexStr		:= ADR(tOilConfig.sData_OilCfgUpd);
						xHexStr2ByteArr.iLenByteWr	:= 7;
						xHexStr2ByteArr.iLenStrRd	:= iOQS_OC_OilCfg_CharSize;

						IF NOT ((iSendMsgCnt = 1) AND (xHexStr2ByteArr.iOffsetStrRd = 0)) THEN
							xHexStr2ByteArr.iOffsetStrRd	:= xHexStr2ByteArr.iOffsetStrRd + 2*xHexStr2ByteArr.iLenByteWr;
						END_IF;
						xHexStr2ByteArr();

						IF (UINT_TO_INT(iOQS_OC_OilCfg_CharSize) - UINT_TO_INT(xHexStr2ByteArr.iOffsetStrRd)) > 14 THEN
							tDataSend_OC[0] := tOilCfgWrite_SendB0_OC[iSendMsgCnt];
						ELSE
							tDataSend_OC[0] := 16#0B;
						END_IF;
					END_IF;
				END_IF;
				(*----------------------------- END CONFIG OIL ----------------------------*)

			_READ_CONFIG:
				(*--------------------------- BEGIN READ CONFIG ---------------------------*)
				(* oil type reconfiguration *)
				(* read oil type configuration *)
				IF iSendMsgCnt = 0 THEN
					tDataSend_OC	:= tOilCfgRead_Send_OC;
					bSend_OC		:= TRUE;
				ELSE
					IF bAck_OC THEN
						bSend_OC	:= TRUE;
						bAck_OC		:= FALSE;
					END_IF;
				END_IF;
				tDataSend_OC[0]		:= tOilCfgRead_SendB0_OC[iSendMsgCnt];
				(*---------------------------- END READ CONFIG ----------------------------*)

		END_CASE;
	END_IF;

	xCANwrite_OQS_OC.enable	:= bSend_OC;
	xCANwrite_OQS_OC();

	(*---------------------------- PROCESS DATA REQUEST ----------------------------*)
	IF xCANwrite_OQS_OC.enable AND (xCANwrite_OQS_OC.status = 0) THEN
		bSend_OC	:=	FALSE;
	END_IF;
	(*---------------------------- PROCESS DATA REQUEST ----------------------------*)

	xTON_OQS_OC_WriteCommInterrupt(IN:= xCANwrite_OQS_OC.status <> 0, PT:= T#10s);	// write communication outage
	(*=================================================================================*)

	(*=============================== CAN READ COMMANDS ===============================*)
	xCANread_OQS_OC.us_ident	:= IN_AG.iCAN_OQS_OC_us_ident;
	xCANread_OQS_OC.can_id		:= iRecMsgID_OC;
	xCANread_OQS_OC.data_adr	:= ADR(tDataRec_OC);

	IF iOQS_OC_ComState <> iOQS_OC_ComStateOld THEN
		bReceive_OC	:= FALSE;
	ELSE
		bReceive_OC	:= TRUE;
	END_IF;
	iOQS_OC_ComStateOld	:=	iOQS_OC_ComState;

	xCANread_OQS_OC.enable	:= bReceive_OC;
	xCANread_OQS_OC();

	IF xCANread_OQS_OC.enable AND (xCANread_OQS_OC.status = 0) THEN
		CASE iOQS_OC_ComState OF
			_READ_DATA:
				(*---------------------------- PROCESS DATA ----------------------------*)
				iReceiveID_OC	:=	SHL(BYTE_TO_UDINT(tDataRec_OC[0]), 24)
								+	SHL(BYTE_TO_UDINT(tDataRec_OC[1]), 16)
								+	SHL(BYTE_TO_UDINT(tDataRec_OC[2]), 8)
								+		BYTE_TO_UDINT(tDataRec_OC[3]);

				CASE iSendMsgCnt OF
					1:	bAck_OC	:=	(iReceiveID_OC = iID_OC_OilT);
					2:	bAck_OC	:=	(iReceiveID_OC = iID_OC_SensorT);
					3:	bAck_OC	:=	(iReceiveID_OC = iID_OC_OilCond);
					4:	bAck_OC	:=	(iReceiveID_OC = iID_OC_ErrStatus);
				ELSE	bAck_OC	:=	FALSE;
				END_CASE;

				IF bAck_OC THEN
					iSendMsgCnt	:= iSendMsgCnt + 1;
					IF iSendMsgCnt > 4 THEN
						iSendMsgCnt	:= 1;
					END_IF;
				END_IF;

				CASE iReceiveID_OC OF
					iID_OC_OilT:
						iT_Oil_OQS_OC	:=	SHL(BYTE_TO_UDINT(tDataRec_OC[7]), 24)
										+	SHL(BYTE_TO_UDINT(tDataRec_OC[6]), 16)
										+	SHL(BYTE_TO_UDINT(tDataRec_OC[5]), 8)
										+		BYTE_TO_UDINT(tDataRec_OC[4]);
						brsmemcpy(pDest:= ADR(MM2VIS.rT_Oil_OQS_OC), pSrc:= ADR(iT_Oil_OQS_OC), length:= 4);

					iID_OC_SensorT:
						iT_Sensor_OQS_OC	:=	SHL(BYTE_TO_UDINT(tDataRec_OC[7]), 24)
											+	SHL(BYTE_TO_UDINT(tDataRec_OC[6]), 16)
											+	SHL(BYTE_TO_UDINT(tDataRec_OC[5]), 8)
											+		BYTE_TO_UDINT(tDataRec_OC[4]);
						brsmemcpy(pDest:= ADR(MM2VIS.rT_Sensor_OQS_OC), pSrc:= ADR(iT_Sensor_OQS_OC), length:= 4);

					iID_OC_OilCond:
						iOilCond_OQS_OC	:=	SHL(BYTE_TO_UDINT(tDataRec_OC[7]), 24)
										+	SHL(BYTE_TO_UDINT(tDataRec_OC[6]), 16)
										+	SHL(BYTE_TO_UDINT(tDataRec_OC[5]), 8)
										+		BYTE_TO_UDINT(tDataRec_OC[4]);
						brsmemcpy(pDest:= ADR(rOilCond_OQS_OC), pSrc:= ADR(iOilCond_OQS_OC), length:= 4);
						rOilCond_OQS_OC	:=	rOilCond_OQS_OC / 100;										// Oil condition value convert to fraction instead of %

					iID_OC_ErrStatus:
						iErrStatus_OQS_OC :=	BYTE_TO_USINT(tDataRec_OC[4]);
				END_CASE;
				(*---------------------------- PROCESS DATA ----------------------------*)

			_CONFIG_OIL:
				(*---------------------- WAIT FOR ACKNOWLEDGEMENT ----------------------*)
				bAck_OC	:=	(brsmemcmp(pMem1:= ADR(tOilCfgWrite_RecB0_OC[iSendMsgCnt]), pMem2:= ADR(tDataRec_OC[0]), length:= 1) = 0)
						AND	(brsmemcmp(pMem1:= ADR(tOilCfgWrite_Rec_OC[1]), pMem2:= ADR(tDataRec_OC[1]), length:= 3) = 0);

				IF bAck_OC THEN
					iSendMsgCnt	:=	iSendMsgCnt + 1;
					IF iSendMsgCnt > 2 THEN
						iSendMsgCnt	:= 1;
					END_IF;

					IF (UINT_TO_INT(iOQS_OC_OilCfg_CharSize) - UINT_TO_INT(xHexStr2ByteArr.iOffsetStrRd)) < 14 THEN
						iOQS_OC_ComState	:=	_READ_CONFIG;
					END_IF;
				END_IF;
				(*---------------------- WAIT FOR ACKNOWLEDGEMENT ----------------------*)

			_READ_CONFIG:
				(*------------------------ READ OIL CONFIG DATA ------------------------*)
				IF iSendMsgCnt = 0 THEN
					bAck_OC	:=	(brsmemcmp(pMem1:= ADR(tOilCfgRead_RecB0_OC[iSendMsgCnt]), pMem2:= ADR(tDataRec_OC[0]), length:= 1) = 0)
							AND	(brsmemcmp(pMem1:= ADR(tOilCfgRead_Rec_OC[1]), pMem2:= ADR(tDataRec_OC[1]), length:= 7) = 0);

					xByteArr2HexStr.iOffsetByteRd	:= 0;
					xByteArr2HexStr.iOffsetStrWr	:= 0;
				ELSE
					bAck_OC	:=	(brsmemcmp(pMem1:= ADR(tOilCfgRead_RecB0_OC[iSendMsgCnt]), pMem2:= ADR(tDataRec_OC[0]), length:= 1) = 0);

					IF bAck_OC THEN
						xByteArr2HexStr.pHexStr			:= ADR(tOilConfig.sData_OilCfgActive);
						xByteArr2HexStr.pByteArray		:= ADR(tDataRec_OC[1]);
						xByteArr2HexStr.iLenByteRd		:= 7;
						xByteArr2HexStr.iLenStrWr		:= iOQS_OC_OilSerialNr_CharSize;
						xByteArr2HexStr.iOffsetByteRd	:= 0;
						IF NOT ((iSendMsgCnt = 1) AND (xByteArr2HexStr.iOffsetStrWr = 0)) THEN
							xByteArr2HexStr.iOffsetStrWr	:= xByteArr2HexStr.iOffsetStrWr + 2*xByteArr2HexStr.iLenByteRd;
						END_IF;
						xByteArr2HexStr();
					END_IF;
				END_IF;

				IF bAck_OC THEN
					iSendMsgCnt	:=	iSendMsgCnt + 1;
					IF iSendMsgCnt > 2 THEN
						iSendMsgCnt	:= 1;
					END_IF;

					IF UINT_TO_INT(iOQS_OC_OilSerialNr_CharSize) - UINT_TO_INT(xByteArr2HexStr.iOffsetStrWr) <= 14 THEN
						iOQS_OC_ComState	:= _READ_DATA;

						IF 		tOilConfig.sData_OilCfgActive = sStdOilSerialNr[1] THEN	MM2VIS.iOQS_OC_OilTypeIdx	:=	1;
						ELSIF	tOilConfig.sData_OilCfgActive = sStdOilSerialNr[2] THEN	MM2VIS.iOQS_OC_OilTypeIdx	:=	2;
						ELSE															MM2VIS.iOQS_OC_OilTypeIdx	:=	0;
						END_IF;
					END_IF;
				END_IF;
				(*------------------------ READ OIL CONFIG DATA ------------------------*)
		END_CASE;
	ELSE
		bAck_OC	:=	FALSE;
	END_IF;

	xTON_AckMissing(IN:= NOT bAck_OC, PT:= T#5s);
	IF xTON_AckMissing.Q THEN
		iOQS_OC_ComState	:=	_READ_DATA;		// return to read state if acknowledgement is not registered on time
	END_IF;

	xTON_OQS_OC_ReadCommInterrupt(IN:= xCANread_OQS_OC.status <> 0, PT:= T#10s);	// read communication outage
	(*=================================================================================*)

	(* generate MSF warning *)
	xTON_OQS_OC_ValueErr(IN:= (rOilCond_OQS_OC < -0.2) OR (rOilCond_OQS_OC > 0.6), PT:= T#10s);

	bAMM_OQS_OC_MSF			:=	xTON_OQS_OC_ReadCommInterrupt.Q
							OR	xTON_OQS_OC_WriteCommInterrupt.Q
							OR	xTON_OQS_OC_ValueErr.Q
							OR	(iErrStatus_OQS_OC <> 0);

	(*_READ_CONFIG when measure signal failure is reset*)
	xF_TRIG_OQS_OC_MSFOff(CLK:= (bAMM_OQS_OC_MSF));
	IF xF_TRIG_OQS_OC_MSFOff.Q THEN
		iOQS_OC_ComState := _READ_CONFIG;
	END_IF;

	(*Update Old Oil Quality status*)
	IF NOT bAMM_OQS_OC_MSF AND (iOQS_OC_Status <> _iMeasSignalFailure) THEN
		iOQS_OC_StatusOld	:=	iOQS_OC_Status;
	END_IF;

	(* signal conditioning *)
	(* oil quality signal value scaling *)
	xLCRScal_OilQual_OQS_OC.x		:=	rOilCond_OQS_OC;
	xLCRScal_OilQual_OQS_OC.x1		:=	Para.rOQS_OC_ScalAgedOil;
	xLCRScal_OilQual_OQS_OC.x2		:=	Para.rOQS_OC_ScalFreshOil;
	xLCRScal_OilQual_OQS_OC.y1		:=	0.0;
	xLCRScal_OilQual_OQS_OC.y2		:=	1.0;
	xLCRScal_OilQual_OQS_OC();
	rOilQual_OQS_OC					:=	LIMIT(-99.999, xLCRScal_OilQual_OQS_OC.y, 1.0);	// open end towards negative quality values

	MM2VIS.rOilCond_OQS_OC_Unfilt	:=	rOilCond_OQS_OC;
	MM2VIS.rOilQual_OQS_OC_Unfilt	:=	rOilQual_OQS_OC;

	(* filtering *)
	xGR_MAXR_T_Oil_OQS_OC(In:= MM2VIS.rT_Oil_OQS_OC, Gw:= Para.rT_OQS_LimLo, Hy:= 2.0);
	IF xGR_MAXR_T_Oil_OQS_OC.Q AND IN_AG.tEng_Run.Do THEN				// only log sensor values if oil temperature above threshold temperature - else freeze values
		xFILTER_OilCond_OQS_OC(In:= rOilCond_OQS_OC, Filter:= 6000);	// 10min filter time const. with 100ms cycle time
	END_IF;
	xLCRScal_OilQual_OQS_OC(x	:=	xFILTER_OilCond_OQS_OC.Out);
	MM2VIS.rOilQual_OQS_OC		:=	LIMIT(-99.999, xLCRScal_OilQual_OQS_OC.y, 1.0);	// open end towards negative quality values

	xTON_EngRun_1h(IN:= IN_AG.tEng_Run.Do, PT:= T#1h);

	(* tendency evaluation *)
	xTON_SecondTick(IN := NOT xTON_SecondTick.Q, PT := T#750ms);	// 750ms + 2 cycles = 950ms -> produces 1s tick due to 100ms sampling rate
	rOilQual_OQS_OC_1sSum := rOilQual_OQS_OC_1sSum + MM2VIS.rOilQual_OQS_OC;

	IF xTON_SecondTick.Q THEN
		rOilQual_OQS_OC_1sAvg		:=	rOilQual_OQS_OC_1sSum / 10;
		rOilQual_OQS_OC_1sSum		:=	0.0;
	END_IF;

	IF NOT bAMM_OQS_OC_MSF THEN
		xCTD_MinuteTick(CD:= xTON_SecondTick.Q, LOAD:= xCTD_MinuteTick.Q, PV:= 60);
		IF xTON_SecondTick.Q THEN
			rOilQual_OQS_OC_1mSum		:=	rOilQual_OQS_OC_1mSum + rOilQual_OQS_OC_1sAvg;
		END_IF;
		IF xCTD_MinuteTick.Q THEN
			rOilQual_OQS_OC_1mAvg		:=	rOilQual_OQS_OC_1mSum / 60;
			rOilQual_OQS_OC_1mSum		:=	0.0;
		END_IF;

		xCTD_HourTick(CD:= xCTD_MinuteTick.Q, LOAD:= xCTD_HourTick.Q, PV:= 60);
		IF xCTD_MinuteTick.Q THEN
			rOilQual_OQS_OC_1hSum		:=	rOilQual_OQS_OC_1hSum + rOilQual_OQS_OC_1mAvg;
		END_IF;
		IF xCTD_HourTick.Q THEN
			rOilQual_OQS_OC_1hAvg		:=	rOilQual_OQS_OC_1hSum / 60;
			rOilQual_OQS_OC_1hSum		:=	0.0;
		END_IF;

		IF xGR_MAXR_T_Oil_OQS_OC.Q AND xTON_EngRun_1h.Q THEN
			IF xCTD_HourTick.Q THEN
				IF (rOilQual_OQS_OC_Old > -100.0) THEN
					MM2VIS.rOilQualTendency_OQS_OC	:=	rOQS_OC_alpha * (rOilQual_OQS_OC_1hAvg - rOilQual_OQS_OC_Old) * 100 + (1 - rOQS_OC_alpha) * MM2VIS.rOilQualTendency_OQS_OC;	// % per 100 oph, negative if oil quality decreases
				END_IF;
				rOilQual_OQS_OC_Old					:=	rOilQual_OQS_OC_1hAvg;
			END_IF;
		ELSE
			MM2VIS.rOilQualTendency_OQS_OC			:=	0.0;
			rOilQual_OQS_OC_Old						:=	-999.9;
		END_IF;
	ELSE
		MM2VIS.rOilQualTendency_OQS_OC			:=	0.0;
		rOilQual_OQS_OC_Old						:=	-999.9;
	END_IF;

	(* generate warnings *)
	bOQS_OC_RelMon			:=	xTON_EngRun_1h.Q AND xGR_MAXR_T_Oil_OQS_OC.Q;

	IF xTON_OQS_Status_UsedGood.Q THEN	xGR_MINR_OQS_Status_UsedGood.Hy	:=	0.05;	(* trap oil quality status in hysteresis if value below limit for > 10min *)
	ELSE								xGR_MINR_OQS_Status_UsedGood.Hy	:=	0.0;
	END_IF;
	IF xTON_OilQual_ValueLo.Q THEN		xGR_MINR_OQS_Status_UsedBad.Hy	:=	0.05;
	ELSE								xGR_MINR_OQS_Status_UsedBad.Hy	:=	0.0;
	END_IF;
	IF xTON_OilQual_ValueLo1.Q THEN		xGR_MINR_OQS_Status_Old.Hy		:=	0.05;
	ELSE								xGR_MINR_OQS_Status_Old.Hy		:=	0.0;
	END_IF;

	xGR_MINR_OQS_Status_UsedGood(In:= MM2VIS.rOilQual_OQS_OC,	Gw:= Para.rOilQual_OQS_OC_LimLo + 0.2);
	xGR_MINR_OQS_Status_UsedBad	(In:= MM2VIS.rOilQual_OQS_OC,	Gw:= Para.rOilQual_OQS_OC_LimLo);
	xGR_MINR_OQS_Status_Old		(In:= MM2VIS.rOilQual_OQS_OC,	Gw:= Para.rOilQual_OQS_OC_LimLo1);

	xTON_OQS_Status_UsedGood(IN	:=	xGR_MINR_OQS_Status_UsedGood.Q,	PT:= T#10m);
	xTON_OilQual_ValueLo(IN		:=	xGR_MINR_OQS_Status_UsedBad.Q,	PT:= T#10m);
	bOilQual_ValueLo			:=	xTON_OilQual_ValueLo.Q	AND bOQS_OC_RelMon;
	bAMM_OQS_OC_ValueLo			:=	(EDGEPOS(xTON_OQS_Status_UsedGood.Q) AND bOQS_OC_RelMon)
								OR	bOilQual_ValueLo;										(*W9353 early oil quality warning*)

	xTON_OilQual_ValueLo1(IN	:=	xGR_MINR_OQS_Status_Old.Q,		PT:= T#10m);
	bOilQual_ValueLo1			:=	xTON_OilQual_ValueLo1.Q	AND bOQS_OC_RelMon;
	bAMM_OQS_OC_ValueLo1		:=	bOilQual_ValueLo1;										(*W9354 critical oil quality warning*)

	xTON_OilQualTendency_Hi(IN	:= (MM2VIS.rOilQualTendency_OQS_OC < Para.rOilQualTendency_OQS_OC_LimHi), PT := T#10s);
	bOilQualTendency_Hi			:=	xTON_OilQualTendency_Hi.Q AND bOQS_OC_RelMon;
	bAMM_OQS_OC_TendencyHi		:=	bOilQualTendency_Hi;									(*W9355 early oil qual. tendency warning*)

	xTON_OilQualTendency_Hi1(IN	:= (MM2VIS.rOilQualTendency_OQS_OC < Para.rOilQualTendency_OQS_OC_LimHi1), PT := T#10s);
	bOilQualTendency_Hi1		:=	xTON_OilQualTendency_Hi1.Q AND bOQS_OC_RelMon;
	bAMM_OQS_OC_TendencyHi1		:=	bOilQualTendency_Hi1;									(*W9356 critical oil qual. tendency warning*)

	(* generate oil quality status *)
	xTON_OQS_Status_RecoverUsedGood	(IN:= NOT xGR_MINR_OQS_Status_UsedGood.Q,	PT:= T#2h);
	xTON_OQS_Status_RecoverUsedBad	(IN:= NOT xGR_MINR_OQS_Status_UsedBad.Q,	PT:= T#2h);
	xTON_OQS_Status_RecoverOld		(IN:= NOT xGR_MINR_OQS_Status_Old.Q,		PT:= T#2h);
	xTON_OQS_Status_RecoverMSF		(IN:= NOT bAMM_OQS_OC_MSF,					PT:= T#1m); 	// faster recover process for MSF status

	IF MM2VIS.bMsg9002 THEN
		xTON_OQS_Status_RecoverUsedGood(PT:= T#0s);
		xTON_OQS_Status_RecoverUsedBad(PT:= T#0s);
		xTON_OQS_Status_RecoverOld(PT:= T#0s);
	END_IF;

	IF 		bAMM_OQS_OC_MSF	THEN												iOQS_OC_Status	:=	_iMeasSignalFailure;
	ELSIF	MM2VIS.bMsg9356	THEN												iOQS_OC_Status	:=	_iOilQual_Old;
	ELSIF	MM2VIS.bMsg9355 AND (iOQS_OC_Status <> _iOilQual_Old) THEN			iOQS_OC_Status	:=	_iOilQual_UsedBad;
	END_IF;

	CASE iOQS_OC_Status OF
		_iMeasSignalFailure:
			IF xTON_OQS_Status_RecoverMSF.Q THEN								iOQS_OC_Status	:=	iOQS_OC_StatusOld;
			END_IF;
		_iOilQual_Old:
			IF xTON_OQS_Status_RecoverOld.Q AND NOT MM2VIS.bMsg9356 THEN		iOQS_OC_Status	:=	_iOilQual_UsedBad;
			END_IF;
		_iOilQual_UsedBad:
			IF	bOilQual_ValueLo1 THEN											iOQS_OC_Status	:=	_iOilQual_Old;
			ELSIF xTON_OQS_Status_RecoverUsedBad.Q AND NOT MM2VIS.bMsg9355 THEN	iOQS_OC_Status	:=	_iOilQual_UsedGood;
			END_IF;
		_iOilQual_UsedGood:
			IF	bOilQual_ValueLo THEN											iOQS_OC_Status	:=	_iOilQual_UsedBad;
			ELSIF xTON_OQS_Status_RecoverUsedGood.Q THEN						iOQS_OC_Status	:=	_iOilQual_New;
			END_IF;
		_iOilQual_New:
			IF	xTON_OQS_Status_UsedGood.Q THEN									iOQS_OC_Status	:=	_iOilQual_UsedGood;
			END_IF;
	END_CASE;

	MM2VIS.iOQS_OC_Status_Num	:=	iOQS_OC_Status;
	MM2VIS.iOQS_OC_Status		:=	iIdx_OQS_OC_Status_Colors[iOQS_OC_Status];

	(* manage oil sample interval *)
	IF iOQS_OC_Status =	_iOilQual_New THEN
		bOpMsg_ExtendOilSampleOh	:=	NOT VIS2MM.bOQS_OilSampleOh_Man;
		rOQS_OC_OilSampleMult		:=	2.0;
	ELSE
		bOpMsg_ExtendOilSampleOh	:=	FALSE;
		rOQS_OC_OilSampleMult		:=	1.0;
	END_IF;

	(* oil sample interval depending on oil quality status *)
	MM2VIS.iOQS_OilSampleOh	:=	REAL_TO_DINT(DINT_TO_REAL(Para.iOilSamplingNomOh) * rOQS_OC_OilSampleMult);

	(* adjust remaining time to next sample in case of status change *)
	xR_TRIG_OQS_OC_Status_Dec(CLK:= (iOQS_OC_Status <> _iOilQual_New));
	xR_TRIG_OQS_OC_Status_Inc(CLK:= (iOQS_OC_Status = _iOilQual_New));

	IF NOT VIS2MM.bOQS_OilSampleOh_Man THEN
		IF		xR_TRIG_OQS_OC_Status_Dec.Q THEN	MM2VIS.iCnt_OilSampleOh	:=	MM2VIS.iCnt_OilSampleOh/2;
		ELSIF	xR_TRIG_OQS_OC_Status_Inc.Q THEN	MM2VIS.iCnt_OilSampleOh	:=	MIN(MM2VIS.iCnt_OilSampleOh*2, MM2VIS.iOQS_OilSampleOh);
		END_IF;
	END_IF;

ELSE
	(* reset vars *)
	xCANwrite_OQS_OC(enable:= FALSE);
	xCANread_OQS_OC(enable:= FALSE);
	xTON_DataSend_ReqTick(IN:= FALSE);
	xTON_SecondTick(IN:= FALSE);
	xCTD_MinuteTick(LOAD:= TRUE);
	xCTD_HourTick(LOAD:= TRUE);
	xTON_EngRun_1h(IN:= FALSE);
	xTON_OQS_OC_WriteCommInterrupt(IN:= FALSE);
	xTON_OQS_OC_ReadCommInterrupt(IN:= FALSE);
	xTON_OQS_OC_ValueErr(IN:= FALSE);
	iErrStatus_OQS_OC := 0;
	MM2VIS.iOQS_OilSampleOh		:=	VIS2MM.iOilSampleOh;	(* default from manual setting *)
	rOQS_OC_OilSampleMult		:=	1.0;
	VIS2MM.bOQS_OilSampleOh_Man	:=	TRUE;
	xTON_OQS_Status_UsedGood(IN:= FALSE);
	xTON_OilQual_ValueLo(IN:= FALSE);
	xTON_OilQual_ValueLo1(IN:= FALSE);
	xTON_OilQualTendency_Hi(IN:= FALSE);
	xTON_OilQualTendency_Hi1(IN:= FALSE);
	xTON_OQS_Status_RecoverUsedGood(IN:= FALSE);
	xTON_OQS_Status_RecoverUsedBad(IN:= FALSE);
	xTON_OQS_Status_RecoverOld(IN:= FALSE);
	xTON_OQS_Status_RecoverMSF(IN:= FALSE);

	(* reset warnings *)
	bAMM_OQS_OC_ValueLo			:=	FALSE;
	bAMM_OQS_OC_ValueLo1		:=	FALSE;
	bAMM_OQS_OC_TendencyHi		:=	FALSE;
	bAMM_OQS_OC_TendencyHi1		:=	FALSE;
	bAMM_OQS_OC_MSF				:=	FALSE;
	bOpMsg_ExtendOilSampleOh	:=	FALSE;
END_IF;

	(*----------------------------------------------------------------------------------------*)
	(*========== BEGIN SAVE OIL QUALITY SENSOR OIL TYPE CONFIG IN PERMANENT MEMORY ===========*)

	(* 10 seconds timer *)
	xTON_WritePMEM(IN := NOT xTON_WritePMEM.Q, PT:= T#10s);
	xTON_BlockMinFileAge(IN := bBlock_MinFileAge, PT:= T#10m);
	IF xTON_BlockMinFileAge.Q THEN	bBlock_MinFileAge := FALSE; END_IF;

	(* every 10 seconds or at write once the parameter values are copied to the structure pm *)
	IF xTON_WritePMEM.Q OR write_once THEN
		(* ------------- V4.11 ---------------- *)
		pmOQS.sData_OilCfgActive	:= tOilConfig.sData_OilCfgActive;	(* copy parameter value to structure pm *)
		pmOQS.sData_OilCfgUpd		:= tOilConfig.sData_OilCfgUpd;		(* ----------------- " ---------------- *)
	END_IF;

	(* cyclic calculation of parameter checksum	*)
	IF xTON_WritePMEM.Q THEN
		ulChecksum := 0;
		FOR ulPMPointer := ADR(pmOQS) TO (ADR(pmOQS) + pm_len - SIZEOF(ulChkValue)) DO
			memcpy(ADR(ulChkValue), ulPMPointer, SIZEOF(ulChkValue));
			ulChecksum := (ulChecksum XOR ulChkValue)+ulChkValue;
		END_FOR;
		IF ulChecksumOld <> ulChecksum THEN					(* if checksum has changed 		*)
			ulChecksumOld := ulChecksum;					(* save last checksum value		*)
			bWriteDataObj := TRUE;							(* set flag for write checksum	*)
		END_IF;
	END_IF;

	(* write structure pm to the permanent memory module *)
	IF ( (bWriteDataObj AND NOT bBlock_MinFileAge) OR write_once ) THEN
		DatObjWrite_01();									(* run data object write fub 					*)
		IF DatObjWrite_01.status <> ERR_FUB_BUSY THEN		(* wait if data object write fub is busy 		*)
			bWriteDataObj 	:= FALSE;						(* reset data object write flag					*)
			write_once 		:= FALSE;						(* reset write_once flag 						*)
			iPM_WriteCnt 	:= iPM_WriteCnt + 1;			(* counter for done data object module writes	*)
			IF OUT_AG.tAG2PB.iPermStatus >=0 THEN 												(* new V4.06: if not already on error state, then transmit this perm status info *)
				OUT_AG.tAG2PB.iPermStatus := LIMIT(2, OUT_AG.tAG2PB.iPermStatus + 1, 999);		(* new V4.06: transmit OK= positive perm status info *)
				IF OUT_AG.tAG2PB.iPermStatus = 999 THEN OUT_AG.tAG2PB.iPermStatus := 2; END_IF;	(* new V4.06: transmit OK= positive perm status info *)
				OUT_AG.tAG2PB.bPermSetupOk := TRUE;												(* new V4.06: transmit perm status info *)
			END_IF;
			IF DatObjWrite_01.status = ERR_NOERROR THEN		(* if status = NO ERROR -> block further write requests for 10min to avoid CF wear down	*)
				bBlock_MinFileAge := TRUE;
			ELSE											(* if error status not no error 				*)
				pm_Error := 3005;  //:= 4;					(* set data object write error state			*)
			END_IF;
		END_IF;
	END_IF;

	(* set RPS warning if no access to SysRom file is possible *)
	TON_WarnDelay(IN := pm_Error > 0 , PT:= T#15s);
	IF TON_WarnDelay.Q AND (OUT_AG.tAG2PB.iPermStatus >= 0) THEN 	OUT_AG.tAG2PB.iPermStatus := LIMIT(-999999,-UINT_TO_DINT(pm_Error) ,-1);	END_IF;	(* new V4.06: transmit error as negative perm status info *)
	IF (OUT_AG.tAG2PB.iPermStatus < 0) THEN 	OUT_AG.tAG2PB.bPermSetupOk := FALSE;	END_IF;		(* No reset of error bit - every error needs reboot *)		(* new V4.06: transmit perm status info *)

	(*=========== END SAVE OIL QUALITY SENSOR OIL TYPE CONFIG IN PERMANENT MEMORY ============*)

END_PROGRAM
```

#### OilQsensInit.st
```iecst
(*******************************************************************************
AGGR: Oil condition monitoring (init)

This code is confidential and proprietary to the INNIO Company.
It may not be used in any form, or reproduced in any manner, without the express
written permission of the INNIO Company.
Copyright, INNIO Company, 2019

- scale the analog input signals
- supervise the analog signals
- counter handling

Customized modifications: -
------------------------

History:
-------
V0.01	04-05-2010	Waldhart, generated
V4.11.0	05.11.2021	Schmid		new oil quality sensor with CAN readout added
V4.11.1	12.10.2022	Bacci		oil quality sensor modification in accordance with TANDELTA firmware 4.03

Instructions for use:
--------------------
-

Outstandings:
------------
-
*******************************************************************************)

PROGRAM _INIT

	bReceive_OC			:= TRUE;
	bSend_OC			:= TRUE;
	bAck_OC				:= FALSE;
	iOQS_OC_ComState	:= _READ_CONFIG; // to get the oil configuration when the PLC starts
	iOQS_OC_ComStateOld	:= _READ_CONFIG; // to get the oil configuration when the PLC starts

	iSendMsgID_OC		:= 16#600 + iSensorID_OC;
	iRecMsgID_OC		:= 16#580 + iSensorID_OC;
	iSendMsgCnt			:= 0;

	tDataSend_OC[0]	:= 16#40;
	tDataSend_OC[1]	:= 16#30;
	tDataSend_OC[2]	:= 16#61;
	tDataSend_OC[3]	:= 16#01;
	tDataSend_OC[4]	:= 16#00;
	tDataSend_OC[5]	:= 16#00;
	tDataSend_OC[6]	:= 16#00;
	tDataSend_OC[7]	:= 16#00;
	iDataLength_OC	:= 8;

	rOilQual_OQS_OC_Old		:= -999.9;
	rOilQual_OQS_OC_1mAvg	:= -999.9;
	rOilQual_OQS_OC_1hAvg	:= -999.9;
	rOQS_OC_alpha			:= 0.0198;
	iOQS_OC_Status			:= _iOilQual_New;
	iOQS_OC_StatusOld		:= _iOilQual_New;
	xR_TRIG_OQS_OC_Status_Dec(CLK:= (iOQS_OC_Status <> _iOilQual_New));	// call once in init to avoid status change detection at PLC start up
	xR_TRIG_OQS_OC_Status_Inc(CLK:= (iOQS_OC_Status = _iOilQual_New));	// call once in init to avoid status change detection at PLC start up

	(* default oil type configuration strings *)
	FOR idxTyp := 1 TO iNum_StdOilCfg DO	// default oil type
		xHexStr2ByteArr.pHexStr			:=	ADR(sStdOilCfg[idxTyp]);
		xHexStr2ByteArr.pByteArray		:=	ADR(tStdOilCfg[idxTyp,1]);
		xHexStr2ByteArr.iLenByteWr		:=	iOQS_OC_OilCfg_ByteSize;
		xHexStr2ByteArr.iLenStrRd		:=	iOQS_OC_OilCfg_CharSize;
		xHexStr2ByteArr.iOffsetStrRd	:=	0;
		xHexStr2ByteArr();
	END_FOR;

	(*================ BEGIN PERMANENT DATA MODULE FOR OIL TYPE CONFIG STRING ================*)
	(* set some init parameters *)
	xTON_WritePMEM(IN := FALSE, PT:= T#10s);					(* reset used timer function blocks 		*)

	pm_Error 	:= ERR_NOERROR;								(* reset permanent memory error	status			*)
	write_once 	:= FALSE;				 					(* reset flag for write permanent memory once	*)
	pm_len 		:= SIZEOF(pmOQS);							(* define data length of permenent memory		*)
	strcpy(ADR(ModulName),ADR('AuxiliariesGeneral::OQS_perm'));		(* define name of permanent memory data module	*)

	(* check for existing permanent memory data module	*)
	DatObjInfo_01.enable:= TRUE;							(* enable FUB									*)
	DatObjInfo_01.pName := ADR(ModulName);					(* set permanent memory data module name 		*)
	DatObjInfo_01();										(* run data object info FUB						*)

	(* check error status of data object info FUB	*)
	IF DatObjInfo_01.status = ERR_NOERROR THEN				(* if no error	--> permanent memory data module exists	*)
		pm_id 	:= DatObjInfo_01.ident;						(* copy permanent memory data module ident			*)
		pm_p 	:= DatObjInfo_01.pDatObjMem;				(* copy permanent memory data module memory adres	*)
	ELSE
		bCreateDataObj := TRUE;								(* set flag for create new data object	*)
		pm_Error := 3001;									(* set permanent memory error status	*)
	END_IF;

	(* check length of parameter struct with length of data object *)

	CASE DatObjInfo_01.len OF
	792:	perm_oqs_vers  := 411;							(* 792 = length of perm_par V4.11 *)
			OUT_AG.tAG2PB.iPermStatus := OUT_AG.tAG2PB.iPermStatus + perm_oqs_vers	;	(* new V4.06: transmit perm status info *)
		//  OUT_AG.tAG2PB.bPermSetupOk := TRUE	;				(* new V4.06: transmit perm status info *)

			(* insert new perm_par Version here
			(* 		   bCreateDataObj := TRUE;						(* set flag for create new data object	*)
			(* xxxx:   perm_oqs_vers  := yyy;						(* xxxx = length of perm_par Vy.yy *)

	ELSE
			bCreateDataObj := TRUE;								(* set flag for create new data object	*)
			OUT_AG.tAG2PB.bPermSetupOk := FALSE	;				(* new V4.06: transmit perm status info *)
			OUT_AG.tAG2PB.iPermStatus := OUT_AG.tAG2PB.iPermStatus  - 1000 ;			(*Perm Error*)
	END_CASE;

	(* if permanent memory data module exist read data and copy to structure pm	*)
	IF pm_Error = ERR_NOERROR THEN							(* permanent memory data module exist 				*)
		DatObjRead_01.enable 		:= TRUE;				(* enable read permanent memory module data 		*)
		DatObjRead_01.ident 		:= pm_id;				(* set identifier of permanent memory data module	*)
		DatObjRead_01.Offset 		:= 0;					(* start at memory offest zero 						*)
		DatObjRead_01.pDestination 	:= ADR(pmOQS);			(* set permanent data destination adress			*)
		DatObjRead_01.len 			:= DatObjInfo_01.len;	(* set length of permanent data module				*)

		REPEAT	(* repeat until data of permanent memory data module have been read *)
			DatObjRead_01();								(* FUB read data from permanent data module 		*)
			UNTIL	DatObjRead_01.status <> ERR_FUB_BUSY	(* wait if FUB is busy 	*)
		END_REPEAT;

		IF DatObjRead_01.status <> ERR_NOERROR THEN			(* if status of read permanent data moduel is not OK 	*)
			pm_Error :=	3002;								(* set permanent memory error status					*)
		END_IF;
	END_IF;

	(* if permanent memory data module exist --> copy data from structure pm to program parameter *)
	IF pm_Error = ERR_NOERROR THEN

		(* ------------- V4.11 ---------------- *)
		tOilConfig.sData_OilCfgActive	:= pmOQS.sData_OilCfgActive;
		tOilConfig.sData_OilCfgUpd		:= pmOQS.sData_OilCfgUpd;

		IF OUT_AG.tAG2PB.iPermStatus >= 0 THEN 													(* new V4.06: transmit perm status info *)
			OUT_AG.tAG2PB.iPermStatus	:= LIMIT(2, OUT_AG.tAG2PB.iPermStatus + pm_len, 999999);	(* new V4.06: transmit perm status info *)
			OUT_AG.tAG2PB.bPermSetupOk	:= TRUE;												(* new V4.06: transmit perm status info *)
		END_IF;																					(* new V4.06: transmit perm status info *)
	END_IF;

	(* create new permanent memory data module	*)
	IF bCreateDataObj THEN

		(* try to delete old data module *)
		DatObjDelete_PermMem.enable := TRUE;
		DatObjDelete_PermMem.ident 	:= pm_id;

		REPEAT	(* repeat until delete of permanent memory data module is ready *)
			DatObjDelete_PermMem();						(* FUB for delete permanent memory data module *)
			UNTIL	DatObjDelete_PermMem.status <> ERR_FUB_BUSY		(* wait if FUB is busy 	*)
		END_REPEAT;

		(* create new one *)
		DatObjCreate_01.enable	 := TRUE;				(* enable create permanent memory data module FUB 	*)
		DatObjCreate_01.grp 	 := 0;					(* must to be set to zero							*)
		DatObjCreate_01.pName 	 := ADR(ModulName);		(* set permanent memory data module name 			*)
		DatObjCreate_01.len 	 := pm_len;				(* set length ofpermanent memory data module		*)
		DatObjCreate_01.MemType  := doUSRROM;			(* create permanent memory data module at USERROM	*)
		DatObjCreate_01.Option 	 := 0;					(* cyclic checksum monitoring is on					*)
		DatObjCreate_01.pCpyData := 0;					(* no data will be copied do the perm. mem. data module *)

		pm_Error:= 3003;								(* set permanent memory error status	*)

		REPEAT	(* repeat until generation of permanent memory data module is ready *)
			DatObjCreate_01();							(* FUB for create permanent memory data module 		*)
			UNTIL	DatObjCreate_01.status <> ERR_FUB_BUSY		(* wait if FUB is busy 	*)
		END_REPEAT;

		IF DatObjCreate_01.status = ERR_NOERROR THEN	(* is creation of permanent memory data module OK 	*)
			pm_p 	:= DatObjCreate_01.pDatObjMem;		(* set memory adress of permanent memory data module*)
			pm_id 	:= DatObjCreate_01.ident;			(* set identifier of permanent memory data module 	*)
		ELSE
			pm_Error:= 3004;							(* set permanent memory error status	*)
		END_IF;
	END_IF;

	(* prepare parameter for permanent memory data write in cyclic task *)
	IF pm_Error < 3004 THEN								(* permanent memory data module exist or has been created	*)
		DatObjWrite_01.enable 	:= TRUE;				(* enable permanent memory data module read FUB 	*)
		DatObjWrite_01.ident 	:= pm_id;				(* set identifier of permanent memory data module 	*)
		DatObjWrite_01.Offset 	:= 0;					(* start at memory offest zero 						*)
		DatObjWrite_01.pSource 	:= ADR(pmOQS);			(* set permanent memory data module name 			*)
		DatObjWrite_01.len 		:= pm_len;				(* set length ofpermanent memory data module		*)
	END_IF;

	(* calcualte actual checksum of parameter structure	*)
	ulChecksumOld := 0;									(* reset checksum value *)

	FOR ulPMPointer := ADR(pmOQS) TO (ADR(pmOQS) + pm_len - SIZEOF(ulChkValue)) DO
		memcpy(ADR(ulChkValue), ulPMPointer, SIZEOF(ulChkValue));
		ulChecksumOld := ulChecksumOld XOR ulChkValue;
	END_FOR

	(**Forward Perm Error - new V4.06 *)
	IF (pm_Error > 0) AND (OUT_AG.tAG2PB.iPermStatus >= 0) THEN 	OUT_AG.tAG2PB.iPermStatus := LIMIT(-999999,-UINT_TO_DINT(pm_Error) ,-1)	;	END_IF		(* new V4.06: transmit error as negative perm status info *)
	IF (OUT_AG.tAG2PB.iPermStatus < 0) THEN 	OUT_AG.tAG2PB.bPermSetupOk := FALSE	;	END_IF			(* new V4.06: transmit perm status info *)

	(*================ END PERMANENT DATA MODULE FOR OIL TYPE CONFIG STRING ================*)

END_PROGRAM
```

#### OilQsens.var
```iecst
(********************************************************************
 * COPYRIGHT -- INNIO Company
 ********************************************************************
 * Program: Oilsensor
 * File: Oilsensor.var
 * Author: WeiglCh
 * Created: June 06, 2008
 ********************************************************************
 * Local variables of program Oilsensor
 ********************************************************************)
(*task vars*)
VAR
	bSend_OC : BOOL; (*Boolean flag to send message to sensor*)
	bAck_OC : BOOL; (*Boolean flag from message aknowledged*)
	iDataLength_OC : UDINT; (*Message lenght in byte*)
	iSendMsgID_OC : UDINT; (*ID message send to sensor*)
	iRecMsgID_OC : UDINT; (*ID message receive from sensor*)
	tDataSend_OC : ARRAY[0..7] OF BYTE; (*Data array containing message for sensor*)
	iReceiveID_OC : UDINT; (*Received message Idenfifier*)
	iT_Oil_OQS_OC : UDINT; (*Oil temperature [degC]*)
	iT_Sensor_OQS_OC : UDINT; (*Sensor temperature [degC]*)
	iOilCond_OQS_OC : UDINT; (*Oil condition, loss factor [%]*)
	iErrStatus_OQS_OC : USINT; (*Error status[/]*)
	iSendMsgCnt : UINT; (*Send message counter*)
	rOilCond_OQS_OC : REAL; (*Oil condition, loss factor [/]*)
	xFILTER_OilCond_OQS_OC : FILTER_R; (*Oil condition filter function*)
	rOilQual_OQS_OC_Old : REAL; (*Old 1h average oil quality*)
	rOilQual_OQS_OC_1sSum : REAL; (*1s sum of oil quality values*)
	rOilQual_OQS_OC_1sAvg : REAL; (*1s average oil quality*)
	xTON_SecondTick : TON; (*TON FUB for 1s tick*)
	xCTD_MinuteTick : CTD; (*CTD FUB for 1min tick*)
	rOilQual_OQS_OC_1mSum : REAL; (*1min sum of oil quality values*)
	rOilQual_OQS_OC_1mAvg : REAL; (*1min average oil quality*)
	rOilQual_OQS_OC_1hSum : REAL; (*1h sum of oil quality values*)
	rOilQual_OQS_OC_1hAvg : REAL; (*1h average oil quality*)
	xCTD_HourTick : CTD; (*CTD FUB for 1h tick*)
	xGR_MAXR_T_Oil_OQS_OC : GR_MAXR; (*Maximum limit monitoring with hysteresis FUB for oil temperature*)
	xCANread_OQS_OC : CANread; (*CAN read FUB between PLC and sensor*)
	xCANwrite_OQS_OC : CANwrite; (*CAN write FUB between PLC and sensor*)
	bReceive_OC : BOOL; (*Boolean flag to receive message from sensor*)
	tDataRec_OC : ARRAY[0..7] OF BYTE; (*Data array containing message from sensor*)
	xTON_DataSend_ReqTick : TON;
	rOQS_OC_alpha : REAL; (*Weighting factor*)
	bOQS_OC_RelMon : BOOL; (*Boolean variable to allow oil monitoring with oil quality sensor*)
	xTON_EngRun_1h : TON; (*TON FUB for 1h of running engine*)
	xLCRScal_OilQual_OQS_OC : LCRScal; (*Scaling FUB for Oil quality*)
	rOilQual_OQS_OC : REAL; (*Oil quality rescaled*)
	xTON_OQS_OC_WriteCommInterrupt : TON; (*TON FUB for write command interrupt*)
	xTON_OQS_OC_ReadCommInterrupt : TON; (*TON FUB for read command interrupt*)
	xTON_OQS_OC_ValueErr : TON; (*TON FUB for read command interrupt*)
	tOilConfig : tOQS_OC_OilConfig; (*Structure containing the updated and active oil configuration*)
	tStdOilCfg : ARRAY[1..2,0..iOQS_OC_OilCfg_ByteSize] OF BYTE; (*Standard oil configurations arrays in byte*)
	idxTyp : UINT; (*Oil configuration index *)
	rOQS_OC_OilSampleMult : REAL; (*Oil sample time interval multiplier*)
	iOQS_OC_Status : USINT; (*Current oil quality status*)
	iOQS_OC_StatusOld : USINT; (*Previous oil quality status*)
	xGR_MINR_OQS_Status_UsedGood : GR_MINR; (*Minimum limit monitoring with hysteresis FUB for oil temperature*)
	xHexStr2ByteArr : HexStr2ByteArr; (*Hex string to byte array FUB converter*)
	xByteArr2HexStr : ByteArr2HexStr; (*Byte array to Hex string FUB converter*)
	iOQS_OC_ComState : UINT; (*Current communication state between the PLC and sensor*)
	iOQS_OC_ComStateOld : UINT; (*Previous communication state between the PLC and sensor*)
	xTON_AckMissing : TON; (*TON FUB for message not aknowledged*)
	xTON_OilQual_ValueLo : TON; (*TON FUB  for used bad oil quality status (lower than 0.4)*)
	xTON_OilQual_ValueLo1 : TON; (*TON FUB  for old oil quality status (lower than 0.2)*)
	xTON_OilQualTendency_Hi : TON; (*TON FUB for oil quality tendency smaller then -0.4*)
	xTON_OilQualTendency_Hi1 : TON; (*TON FUB for oil quality tendency smaller then -0.5*)
	bOilQual_ValueLo : BOOL; (*Boolean variable to identify bad oil quality status (lower than 0.4)*)
	bOilQual_ValueLo1 : BOOL; (*Boolean variable to identify bad oil quality status (lower than 0.2)*)
	bOilQualTendency_Hi : BOOL; (*Boolean variable to identify bad oil quality status (lower than 0.4)*)
	bOilQualTendency_Hi1 : BOOL; (*Boolean variable to identify bad oil quality status (lower than 0.4)*)
	xGR_MINR_OQS_Status_UsedBad : GR_MINR; (*Minimum limit monitoring with hysteresis FUB for used bad oil quality status*)
	xGR_MINR_OQS_Status_Old : GR_MINR; (*Minimum limit monitoring with hysteresis FUB for old oil quality status*)
	xTON_OQS_Status_UsedGood : TON; (*TON FUB for used good oil quality status*)
	xTON_OQS_Status_RecoverUsedGood : TON; (*TON FUB for recover from used good oil quality status*)
	xTON_OQS_Status_RecoverUsedBad : TON; (*TON FUB for recover from used bad oil quality status*)
	xTON_OQS_Status_RecoverOld : TON; (*TON FUB for recover from old oil quality status*)
	xTON_OQS_Status_RecoverMSF : TON; (*TON FUB for recover from error message status*)
	xR_TRIG_OQS_OC_Status_Dec : R_TRIG; (*R_TRIG FUB to extend oil sample interval*)
	xR_TRIG_OQS_OC_Status_Inc : R_TRIG; (*R_TRIG FUB to reduce oil sample interval*)
	xF_TRIG_OQS_OC_MSFOff : F_TRIG; (*R_TRIG FUB to reduce oil sample interval*)
END_VAR
(*permanent data module*)
VAR
	write_once : BOOL; (*write permanent memory once *)
	bCreateDataObj : BOOL; (*TRUE=create new data object *)
	bWriteDataObj : BOOL; (*TRUE=write data object module *)
	DatObjCreate_01 : DatObjCreate; (*data object create *)
	DatObjDelete_PermMem : DatObjDelete; (*data object delete *)
	DatObjInfo_01 : DatObjInfo; (*data object info *)
	DatObjRead_01 : DatObjRead; (*data object read *)
	DatObjWrite_01 : DatObjWrite; (*data object write *)
	pmOQS : tOQS_OC_OilConfig; (*permanent memory tags *)
	ModulName : STRING[35]; (*module name of object *)
	xTON_WritePMEM : TON; (*delay write permanent memory *)
	pm_len : UDINT; (*permanent value lenght *)
	pm_p : UDINT; (*permanent value pointer *)
	pm_id : UDINT; (*permanent value identifier *)
	ulChecksumOld : UDINT; (*last vlaue of parameter checksum *)
	ulChecksum : UDINT; (*parameter checksum value *)
	ulPMPointer : UDINT; (*adress of actual checksum value *)
	ulChkValue : UDINT; (*actual value of parameter pointer *)
	pm_Error : UINT; (*permanent value error *)
	perm_oqs_vers : UINT; (*version*)
	ERR_NOERROR : UINT := 0; (* status for no error *)
	TON_WarnDelay : TON; (*V4.06*)
	xTON_BlockMinFileAge : TON;
	bBlock_MinFileAge : BOOL;
	iPM_WriteCnt : UINT; (*data module write counter *)
END_VAR
(*sensor ID and msg constants*)
VAR CONSTANT
	iSensorID_OC : UDINT := 16#1; (*Sensor ID node*)
	iID_OC_OilT : UDINT := 16#43306101; (*ID (first 4 bytes) oil temperature reply message*)
	iID_OC_SensorT : UDINT := 16#43306102; (*ID (first 4 bytes) sensor temperature reply message*)
	iID_OC_OilCond : UDINT := 16#43306103; (*ID (first 4 bytes) oil condition reply message*)
	iID_OC_ErrStatus : UDINT := 16#4F011000; (*ID (first 4 bytes) oil temperature reply message*)
	tDataReq_OC : ARRAY[0..7] OF BYTE := [16#40,16#30,16#61,16#01,4(16#00)]; (*Data request command message *)
	tErrReq_OC : ARRAY[0..7] OF BYTE := [16#40,16#01,16#10,5(16#00)]; (*Error status command message*)
	tOilCfgRead_SendB0_OC : ARRAY[0..2] OF BYTE := [16#40,16#60,16#70]; (*Byte 0  for the different READ_CONFIG command messages*)
	tOilCfgRead_RecB0_OC : ARRAY[0..2] OF BYTE := [16#41,16#00,16#11]; (*Byte 0  for the different READ_CONFIG reply messages*)
	tOilCfgRead_Send_OC : ARRAY[0..7] OF BYTE := [16#40,16#21,16#6F,16#01,4(16#00)]; (*READ_CONFIG command message*)
	tOilCfgRead_Rec_OC : ARRAY[0..7] OF BYTE := [16#41,16#21,16#6F,16#01,16#0E,3(16#00)]; (*READ_CONFIG reply message*)
	tOilCfgWrite_SendB0_OC : ARRAY[0..2] OF BYTE := [16#20,16#00,16#10]; (*Byte 0  for the different READ_CONFIG command messages*)
	tOilCfgWrite_Send_OC : ARRAY[0..7] OF BYTE := [16#21,16#20,16#6F,16#01,16#7C,16#01,2(16#00)]; (*CONFIG_OIL command message*)
	tOilCfgWrite_RecB0_OC : ARRAY[0..2] OF BYTE := [16#60,16#20,16#30]; (*Byte 0  for the different READ_CONFIG command messages*)
	tOilCfgWrite_Rec_OC : ARRAY[0..7] OF BYTE := [16#60,16#20,16#6F,16#01,4(16#00)]; (*CONFIG_OIL reply message*)
	_READ_DATA : UINT := 0; (*_READ_DATA communication status*)
	_CONFIG_OIL : UINT := 1; (*_CONFIG_OIL communication status*)
	_READ_CONFIG : UINT := 2; (*_READ_CONFIG communication status*)
	_iMeasSignalFailure : USINT := 0; (*Signal failure oil quality status*)
	_iOilQual_New : USINT := 1; (*New oil quality status*)
	_iOilQual_UsedGood : USINT := 2; (*Used Good oil quality status*)
	_iOilQual_UsedBad : USINT := 3; (*Used Bad oil quality status*)
	_iOilQual_Old : USINT := 4; (*Old oil quality status*)
	iIdx_OQS_OC_Status_Colors : ARRAY[_iMeasSignalFailure.._iOilQual_Old] OF USINT := [8,2,124,46,51]; (*grey, green, light blue, yellow, red*)
	iNum_StdOilCfg : USINT := 2; (*Number of standard oil configuration*)
	sStdOilCfg : ARRAY[1..iNum_StdOilCfg] OF STRING[iOQS_OC_OilCfg_CharSize] := ['21156BD9252C1542154B5015255E1515151564151515FA3B56251515254915252515003315002115B8AC7A9C15A8154BAF1583B515151515B7151515EFA4B28B151598AC1572921500A0150121157B27B8AF15A1154B9815B78B1515151584151515E4A592B61515B39C15B8B51500AB15022115D875673A141A144B01155DEB15151515E1151415DC25F5541415430E156E4C1500301503211444F0C48D1474144B6414B954141414144C141414D27C5CAE1414986C14CEA31400841404211405FF361E1412144B0C1431081414141406141414CF160A2C1414230E143C2814001A1405211303BD01FF14FF144B001401011414141402131414C9FF01001413FF001303001300FF140621141B9D050B140F144B131406171414141419141414C70E150714140A1114040814000C140721144842202D1435144B3B1422421414141445141414C3323E2514142B38141D2814003014082114309A4F4F3132354B30144F383014141446473020BD20304F30004F3A144B4F0000001409','23EBEC131313EC3DD013E6E6E9E613E6E6EA1313F01313E71313EA13131313EDED0013E6ED0023E1DF131313D1E4D013E9EAE5EC13E8EBE41313E01313E71313E313131313DCD40013EBD80123AAA61313139680D013C2C5B5CF13BDCCB01313D41313B91313AD13131313A39A0013C99E02236D681313135CEDD01383867891137F96741313CB13137B13137013131313645E00138961032344431313133F24D0134F524859134C57471313C613134A131346131313134240001354410423424313131347E3D0133E3E403F133E3E411313C013133F13134113131313444600133E4505235B5C1313136549D013514F564913534B571313BA131354131359131313135E6200134D6006237F821313138D84D013716E776713736A7A1313B113137513137C13131313858A00136C870723AEB1131313C0E5D0139C99A490139F93A81313A51313A21313AB13131313B5BC001396B908233A30303200300AD013C8C800C413C8C82035009D3020C81313321313301330300047C83809']; (*Standard oil configuration*)
	sStdOilSerialNr : ARRAY[1..iNum_StdOilCfg] OF STRING[iOQS_OC_OilSerialNr_CharSize] := ['4732203A30303030303831463530','4732203A30303030303832303530']; (*Standard oil serial number*)
END_VAR
```

#### OilQsens.fun
```iecst
FUNCTION_BLOCK HexStr2ByteArr
	VAR_INPUT
		pHexStr : UDINT;
		iLenStrRd : UINT;
		pByteArray : UDINT;
		iLenByteWr : UINT;
		iOffsetStrRd : UINT;
	END_VAR
	VAR
		idxByte : UINT;
		idxChar : UINT;
		idxRead : UINT;
		iByte : UINT;
		sChar : STRING[1];
		pCurrArrPos : UDINT;
	END_VAR
END_FUNCTION_BLOCK

FUNCTION_BLOCK ByteArr2HexStr
	VAR_INPUT
		pByteArray : UDINT;
		iLenByteRd : UINT;
		pHexStr : UDINT;
		iLenStrWr : UINT;
		iOffsetByteRd : UINT;
		iOffsetStrWr : UINT;
	END_VAR
	VAR
		idxNibble : UINT;
		idxByte : UINT;
		idxRead : UINT;
		iByte : UINT;
		iNibble : UINT;
		sChar : STRING[1];
		pCurrArrPos : UDINT;
	END_VAR
END_FUNCTION_BLOCK
```

#### ConvByteHex.st
```iecst
FUNCTION_BLOCK HexStr2ByteArr
	pCurrArrPos	:= pByteArray;

	FOR idxByte := 0 TO iLenByteWr-1 DO	// selected byte
		iByte	:=	0;
		FOR idxChar	:=	0 TO 1 DO			// selected config string characters
			idxRead	:= idxByte*2 + idxChar + iOffsetStrRd;
			IF idxRead < iLenStrRd THEN
				brsmemcpy(ADR(sChar), pHexStr + idxRead, 1);
			ELSE
				sChar	:=	'';
			END_IF;

			IF 		sChar = '0' THEN	iByte	:=	iByte	+	TRUNC(0	* 16 ** (1-idxChar));
			ELSIF	sChar = '1' THEN	iByte	:=	iByte	+	TRUNC(1	* 16 ** (1-idxChar));
			ELSIF	sChar = '2' THEN	iByte	:=	iByte	+	TRUNC(2	* 16 ** (1-idxChar));
			ELSIF	sChar = '3' THEN	iByte	:=	iByte	+	TRUNC(3	* 16 ** (1-idxChar));
			ELSIF	sChar = '4' THEN	iByte	:=	iByte	+	TRUNC(4	* 16 ** (1-idxChar));
			ELSIF	sChar = '5' THEN	iByte	:=	iByte	+	TRUNC(5	* 16 ** (1-idxChar));
			ELSIF	sChar = '6' THEN	iByte	:=	iByte	+	TRUNC(6	* 16 ** (1-idxChar));
			ELSIF	sChar = '7' THEN	iByte	:=	iByte	+	TRUNC(7	* 16 ** (1-idxChar));
			ELSIF	sChar = '8' THEN	iByte	:=	iByte	+	TRUNC(8	* 16 ** (1-idxChar));
			ELSIF	sChar = '9' THEN	iByte	:=	iByte	+	TRUNC(9	* 16 ** (1-idxChar));
			ELSIF	sChar = 'A' THEN	iByte	:=	iByte	+	TRUNC(10* 16 ** (1-idxChar));
			ELSIF	sChar = 'B' THEN	iByte	:=	iByte	+	TRUNC(11* 16 ** (1-idxChar));
			ELSIF	sChar = 'C' THEN	iByte	:=	iByte	+	TRUNC(12* 16 ** (1-idxChar));
			ELSIF	sChar = 'D' THEN	iByte	:=	iByte	+	TRUNC(13* 16 ** (1-idxChar));
			ELSIF	sChar = 'E' THEN	iByte	:=	iByte	+	TRUNC(14* 16 ** (1-idxChar));
			ELSIF	sChar = 'F' THEN	iByte	:=	iByte	+	TRUNC(15* 16 ** (1-idxChar));
			ELSE						iByte	:=	0;
			END_IF;
		END_FOR;

		IF (pCurrArrPos - pByteArray) < iLenByteWr THEN
			pCurrArrPos	:=	brsmemset(pCurrArrPos, UINT_TO_USINT(iByte), 1);
		END_IF;
	END_FOR;
END_FUNCTION_BLOCK

FUNCTION_BLOCK ByteArr2HexStr
	pCurrArrPos	:= pHexStr + iOffsetStrWr;

	FOR idxByte := 0 TO iLenByteRd-1 DO	// selected byte
		iByte	:=	0;

		idxRead	:= idxByte + iOffsetByteRd;
		IF idxRead < iLenStrWr/2 THEN
			brsmemcpy(ADR(iByte), pByteArray + idxRead, 1);
		ELSE
			iByte	:=	0;
		END_IF;
		FOR idxNibble	:=	0 TO 1 DO			// selected 4 bit (nibble) byte subgroup
			IF idxNibble = 0 THEN
				iNibble	:=	SHR(iByte, 4);
			ELSE
				iNibble	:=	iByte MOD 16;
			END_IF;

			IF 		iNibble = 0		THEN	sChar := '0';
			ELSIF	iNibble = 1		THEN	sChar := '1';
			ELSIF	iNibble = 2		THEN	sChar := '2';
			ELSIF	iNibble = 3		THEN	sChar := '3';
			ELSIF	iNibble = 4		THEN	sChar := '4';
			ELSIF	iNibble = 5		THEN	sChar := '5';
			ELSIF	iNibble = 6		THEN	sChar := '6';
			ELSIF	iNibble = 7		THEN	sChar := '7';
			ELSIF	iNibble = 8		THEN	sChar := '8';
			ELSIF	iNibble = 9		THEN	sChar := '9';
			ELSIF	iNibble = 10	THEN	sChar := 'A';
			ELSIF	iNibble = 11	THEN	sChar := 'B';
			ELSIF	iNibble = 12	THEN	sChar := 'C';
			ELSIF	iNibble = 13	THEN	sChar := 'D';
			ELSIF	iNibble = 14	THEN	sChar := 'E';
			ELSIF	iNibble = 15	THEN	sChar := 'F';
			ELSE							sChar := '0';
			END_IF;

			IF (pCurrArrPos - pHexStr) < iLenStrWr THEN
				pCurrArrPos	:= brsmemcpy(pCurrArrPos, ADR(sChar), 1);
			END_IF;
		END_FOR;
	END_FOR;
END_FUNCTION_BLOCK
```

### Program Logical/AuxiliariesGeneral/FiltUnit (IEC, version 4.11.0) - Oil filter unit

#### FiltUnitCyclic.st - Cyclic code
```iecst
(****************************************************************************************************************************
FiltUnit		Oil filter unit (CYCLIC)

This code is confidential and proprietary to the INNIO Company.
It may not be used in any form, or reproduced in any manner,
without the express written permission of the INNIO Company.
Copyright, INNIO Company, 2019

Customized modifications: -
------------------------

History:
-------
V4.04.00.00		24.05.2016 TinelloM	erstellt
				01.09.2016 TinelloM	Anpassung an Speziupdate
V4.07.00.00		13.05.2019 Schmid	OUT interface OUT_AG.rDPr_OFU_Filt added
V4.09.00.00		05.03.2020 Schmid	oil centrifuge must not run at interval/perm. prelube
V4.11.00.00		21.12.2021 Schmid	pressure before oil centrifuge min warning added

(****************************************************************************************************************************)
PROGRAM _CYCLIC

	IF Para.bOilFiltUnit_Exist AND IN_AG.tPB2MM.bParaSetupOk THEN

		(* monitoring of oilfilter difference pressure *)
		rDPr_OFU_Filt				:= IN_AG.tPr_OFUbFilt.Ai - IN_AG.tPr_OFUaFilt.Ai;

		bAMM_DPr_OFU_Filt_Hi		:= (rDPr_OFU_Filt 	> Para.rDPr_OFU_Filt_LimHi) 				AND				(* W2629 *)
										 Para.bPr_OFUbFilt_Active 	AND  Para.bPr_OFUaFilt_Active  	AND
										IN_AG.tPr_OFUbFilt.GoodQual	AND IN_AG.tPr_OFUaFilt.GoodQual;

		bAMM_DPr_OFU_Filt_HiHi		:= (rDPr_OFU_Filt 	> Para.rDPr_OFU_Filt_LimHi + 2) 			AND	(* +2bar *)	(* W2422 *)
										 Para.bPr_OFUbFilt_Active 	AND  Para.bPr_OFUaFilt_Active  	AND
										IN_AG.tPr_OFUbFilt.GoodQual	AND IN_AG.tPr_OFUaFilt.GoodQual;

		(* monitoring of pressure maximum *)
		bAMM_Pr_OFUbFilt_Hi			:= IN_AG.tPr_OFUbFilt.Ai > Para.rPr_OFUbFilt_Hi	AND								(* W2785 *)
									    Para.bPr_OFUbFilt_Active	AND
									   IN_AG.tPr_OFUbFilt.GoodQual;

		bAMM_Pr_OFUbCentrifuge_Hi	:= IN_AG.tPr_OFUbCentrifuge.Ai > Para.rPr_OFUbCentrifuge_Hi AND					(* W2787 *)
									    Para.bPr_OFUbCentrifuge_Active 	AND
									   IN_AG.tPr_OFUbCentrifuge.GoodQual;

		(* monitoring of pressure minimum *)
		xTON_AMM_Centrifuge_Pr_Lo_MonRel(IN:= OUT_AG.tOFUP_Centrifuge.Do, PT:= T#5m);

		bAMM_Pr_OFUbCentrifuge_Lo	:=	IN_AG.tPr_OFUbCentrifuge.Ai < Para.rPr_OFUbCentrifuge_Lo			(* W9359 *)
									AND	xTON_AMM_Centrifuge_Pr_Lo_MonRel.Q
									AND	Para.bPr_OFUbCentrifuge_Active
									AND IN_AG.tPr_OFUbCentrifuge.GoodQual;

		(* oil pump centrifuge / M.03-P-006 *)
		xTOF_OFUP_Centrifuge_Dem(IN:= bPreLubeDem OR M_DREHZ, PT:= T#10m);
		OUT_AG.tOFUP_Centrifuge.Do	:= bOMSS_MAT					AND					(* panel switch ON *)
									   IN_AG.tOFUP_Centrifuge_CB.Di	AND					(* oil centrifuge circuit breaker OK *)
									   NOT bGnlTrip					AND			 		(* no trip *)
									   IN_AG.tT_EO_Pan.Ai > 70 		AND					(* temp. oil pan > 70°C *)
									   NOT MM2VIS.bMsg2786			AND					(* press. before centrifuge sig. Err *)
									   NOT MM2VIS.bMsg2787			AND					(* press. before centrifuge maximum *)
									   xTOF_OFUP_Centrifuge_Dem.Q;						(* oil pump in operation *)

		(* oil pump oilfilter / M.03-P-007 *)
			xTON_Centrifuge(IN		:= OUT_AG.tOFUP_Centrifuge.Do, PT:= T#2s );

		OUT_AG.tOFUP_Filter.Do		:= xTON_Centrifuge.Q			AND					(* no start of both pumps together *)
									   IN_AG.tOFUP_Filter_CB.Di		AND					(* oilfilter pump circuit breaker OK *)
									   NOT MM2VIS.bMsg2627			AND					(* press. before oil filter sig. Err *)
									   NOT MM2VIS.bMsg2628			AND					(* press. after oil filter sig. Err *)
									   NOT MM2VIS.bMsg2785			AND					(* press. before oil filter maximum *)
									   NOT MM2VIS.bMsg2422;								(* diff press < limit + 2bar *)

	ELSE
		(* reset *)
		bAMM_DPr_OFU_Filt_Hi		:= FALSE;
		bAMM_DPr_OFU_Filt_HiHi		:= FALSE;
		bAMM_Pr_OFUbFilt_Hi			:= FALSE;
		bAMM_Pr_OFUbCentrifuge_Hi	:= FALSE;
		bAMM_Pr_OFUbCentrifuge_Lo	:= FALSE;
		xTON_AMM_Centrifuge_Pr_Lo_MonRel(IN:= FALSE);
		xTOF_OFUP_Centrifuge_Dem(IN:= FALSE);
		xTON_Centrifuge(IN:= FALSE);
		OUT_AG.tOFUP_Centrifuge.Do	:= FALSE;
		OUT_AG.tOFUP_Filter.Do		:= FALSE;
		rDPr_OFU_Filt				:= 0;
	END_IF

	(* VISU *)
	MM2VIS.rPr_OFUbCentrifuge		:= IN_AG.tPr_OFUbCentrifuge.Ai;
	MM2VIS.rPr_OFUaFilt				:= IN_AG.tPr_OFUaFilt.Ai;
	MM2VIS.rPr_OFUbFilt 			:= IN_AG.tPr_OFUbFilt.Ai;
	MM2VIS.rDPr_OFU_Filt			:= rDPr_OFU_Filt;
	MM2VIS.bOFUP_Centrifuge			:= OUT_AG.tOFUP_Centrifuge.Do;
	MM2VIS.bOFUP_Filter				:= OUT_AG.tOFUP_Filter.Do;

	OUT_AG.rDPr_OFU_Filt			:= rDPr_OFU_Filt;

END_PROGRAM
```

#### FiltUnit.var - Local variables
```iecst
VAR
	rDPr_OFU_Filt : REAL := 0; (*oilfilter difference pressure (oil filter unit)*)
	xTON_Centrifuge : TON := (0); (*FuB*)
	xTOF_OFUP_Centrifuge_Dem : TOF;
	xTON_AMM_Centrifuge_Pr_Lo_MonRel : TON;
END_VAR
```

### Program Logical/AuxiliariesGeneral/PermAG (IEC, version 4.14.0) - + PermanentMemory

- PermAGCyclic.st (not readable text: treated as protected, skipped)

- PermAGInit.st (not readable text: treated as protected, skipped)

#### PermAG.var
```iecst
VAR
	pm_Error : UINT;
	write_once : BOOL;
	pm_len : UDINT;
	ModulName : STRING[35];
	DatObjInfo_01 : DatObjInfo;
	pm_id : UDINT;
	pm_p : UDINT;
	bCreateDataObj : BOOL;
	perm_par_vers : UINT;
	DatObjRead_01 : DatObjRead;
	usPMWriteCnt : UINT;
	DatObjDelete_PermMem : DatObjDelete;
	DatObjCreate_01 : DatObjCreate;
	DatObjWrite_01 : DatObjWrite;
	ulChecksumOld : UDINT;
	ulPMPointer : UDINT;
	ulChkValue : UDINT;
	TON_WritePMEM : TON;
	ulChecksum : UDINT;
	bWriteDataObj : BOOL;
END_VAR
VAR CONSTANT
	ERR_NOERROR : UINT := 0;
END_VAR
VAR
	pmm : Perm_AG_Struct;
	TON_WarnDelay : TON := (0);
END_VAR
```

### Program Logical/AuxiliariesGeneral/OilTank (IEC, version 4.12.0) - Oiltank volume for fresh- & waste- oil tank & day tank
